// TwinCAT 3 PLC project Projet_Base
// ProgramVersion: 3.1.4026.12
// CompilerDefines: VISU_USEPROPERTYINFO
// libraries:
//   CmpBitmapPool, * (System)
//   Tc2_ControllerToolbox, * (Beckhoff Automation GmbH)
//   Tc2_ModbusRTU, * (Beckhoff Automation GmbH)
//   Tc2_ModbusSrv, * (Beckhoff Automation GmbH)
//   Tc2_SerialCom, * (Beckhoff Automation GmbH)
//   Tc2_Standard, * (Beckhoff Automation GmbH)
//   Tc2_System, * (Beckhoff Automation GmbH)
//   Tc2_TcpIp, * (Beckhoff Automation GmbH)
//   Tc2_Utilities, * (Beckhoff Automation GmbH)
//   Tc3_Database, * (Beckhoff Automation GmbH)
//   Tc3_Module, * (Beckhoff Automation GmbH)
//   BASIC,3.31,OSCAT
// project tree:
//   00_FunctionsBlocks/Beckhoff/AlarmManagement/ FB_HeartBeatMasterBackup.TcPOU, FUN_Alarms_CSV.TcPOU, FUN_ReadAlarm_CSV.TcPOU, ServerCSV.TcDUT, ServerSms.TcDUT, SMS_Server.TcPOU
//   00_FunctionsBlocks/Beckhoff/Annexesfunction/ FB_RestartService.TcPOU, FUN_ConnectVPN.TcPOU, FUN_DisconnectVPN.TcPOU, FUN_GetPublicIp.TcPOU, FUN_PingHost.TcPOU, PRG_RestartPlc.TcPOU
//   00_FunctionsBlocks/Beckhoff/Communication/IEC104/ E_ComState.TcDUT, FB_IEC104ServerAkuo.TcPOU, GVL_Cst.TcGVL, ST_IEC104AkuoParam.TcDUT
//   00_FunctionsBlocks/Beckhoff/Communication/Mail/ FUN_SendMail.TcPOU, ServerMail.TcDUT
//   00_FunctionsBlocks/Beckhoff/Communication/ModbusRTU/ CheckStruct.TcPOU, FB_ModbusRTU.TcPOU, FB_ReadModbusRTU_V2.TcPOU, Sample_ModbusRTU.TcPOU, Struct_InputRTU.TcDUT
//   00_FunctionsBlocks/Beckhoff/Communication/ModbusTCP/ FB_ModbusRead.TcPOU, FB_ModbusReadCoils.TcPOU, FB_ModbusReadInput.TcPOU, FB_ModbusReadInputRegs.TcPOU, FB_ModbusWrite.TcPOU, FB_ModbusWriteMultipleCoils.TcPOU, FB_ModbusWriteSingleCoil.TcPOU, FB_ModbusWriteSingleRegister.TcPOU
//   00_FunctionsBlocks/Beckhoff/Communication/SMS/ FB_DeleteAllSMS.TcPOU, FB_DeleteSMS.TcPOU, FB_Extract_Num_Mes.TcPOU, FB_Login.TcPOU, FB_ReadSMS.TcPOU, FB_SendSMS.TcPOU, ST_SMSDataSetEntry_Read.TcDUT, ST_SMSDataSetEntry_Send.TcDUT
//   00_FunctionsBlocks/Beckhoff/Database/ CheckConfig.TcPOU, PRG_EpochConverter.TcPOU, PRG_TimestructConverter.TcPOU, St_DataHisto.TcDUT, St_DataHisto_Epoch.TcDUT, UnixTimestamp.TcPOU
//   00_FunctionsBlocks/Beckhoff/Database/Firebird/ Firebird_CreateTables.TcPOU, Firebird_InsertBuffer.TcPOU, Firebird_InsertBuffer_vEpoch.TcPOU, Firebird_ReadAlarms.TcPOU, Firebird_RetrieveHDBID.TcPOU, Firebird_SelectBuffer.TcPOU, Firebird_WriteAlarms.TcPOU, LoggerFirebird.TcDUT, St_AlarmsV2.TcDUT
//   00_FunctionsBlocks/Beckhoff/Database/InfluxDb/ InfluxDb_AlarmsManagement.TcPOU, InfluxDb_ReadValues.TcPOU, InfluxDb_WriteAlarms.TcPOU, InfluxDb_WriteStruct.TcPOU, LoggerInfluxDb.TcDUT, ST_InfluxAlarmsInsert.TcDUT, ST_InfluxAlarmsRetrieve.TcDUT
//   00_FunctionsBlocks/Beckhoff/Database/SQLCe/ FB_SQLExpert_InsertBuffer_1.TcPOU
//   00_FunctionsBlocks/Beckhoff/Database/SQLite/ SQLite_CreateDb_V2_1.TcPOU, SQLite_DeleteConfDb_1.TcPOU
//   00_FunctionsBlocks/Beckhoff/DataProcessing/Compress/ FB_CompressFile.TcPOU, FUN_CompressCSV.TcPOU
//   00_FunctionsBlocks/Beckhoff/DataProcessing/Database/ DataBase_V2.TcPOU, FB_DeleteFile.TcPOU, FB_SQLExpert_InsertBuffer.TcPOU, SQLite_CreateDb_V2.TcPOU, SQLite_DeleteConfDb.TcPOU
//   00_FunctionsBlocks/Beckhoff/DataProcessing/ FB_MergeWordsToFloat.TcPOU, FB_MessageDynamique.TcPOU, FB_SplitFloatToWords.TcPOU, FB_WordsToFloat32MLE.TcPOU, FUN_Transpose.TcPOU, MOYENNE.TcPOU, ReplaceAll.TcPOU, SavePersistent.TcPOU
//   00_FunctionsBlocks/Beckhoff/DataProcessing/ReadFile/ FB_Read.TcPOU, FB_ReadCSV.TcPOU
//   00_FunctionsBlocks/Beckhoff/DataProcessing/WriteFile/ CheckStruct_Alarms.TcPOU, FB_CreateDir_V2.TcPOU, FB_WriteFile.TcPOU, FB_Write_CSV.TcPOU, FUN_CreateDir_CSV.TcPOU, LoggerCSV.TcDUT, ST_Journal.TcDUT, ST_ValuesAlarms.TcDUT, ST_ValuesWrite.TcDUT
//   00_FunctionsBlocks/Beckhoff/Fifo/ FB_CommandAlternate.TcPOU, FB_DBDatasetFifo.TcPOU, FB_DBDatasetFifo_1min.TcPOU, FB_SMSDatasetFifo_Read.TcPOU, FB_SMSDatasetFifo_Send.TcPOU, GVL_Fifo.TcGVL
//   00_FunctionsBlocks/Common/AlarmManagement/ FB_AlarmCodeManager.TcPOU, FB_CheckCommand.TcPOU, FB_CheckSetpt.TcPOU, FB_DetectFixedValue.TcPOU, FB_DetectFlicker.TcPOU, FB_UnknownEvent.TcPOU
//   00_FunctionsBlocks/Common/BoolManagement/ FB_CountNinTimeWindow.TcPOU, FB_TapVariable.TcPOU, FB_Toggle2Tap.TcPOU, FB_WordToArrayOfBool.TcPOU, FB_WriteOnChange.TcPOU, RS_NoReset.TcPOU
//   00_FunctionsBlocks/Common/Ctrl/ FB_PIDRegulation.TcPOU
//   00_FunctionsBlocks/Common/DataProcessing/ FB_Average.TcPOU, FB_CountBitOfWordAtTrue.TcPOU, FB_Integrate.TcPOU, FB_MovingAverage.TcPOU, FB_Ramp.TcPOU, FB_Ramp_Time.TcPOU, FB_Smooth.TcPOU, FB_XorWord.TcPOU, Split.TcPOU, Substring.TcPOU
//   00_FunctionsBlocks/Common/DataProcessing/MergeWord/ FB_ISKRA_T5.TcPOU, FB_ISKRA_T6.TcPOU, FB_MergeWordsToDint.TcPOU, FB_MergeWordsToUint.TcPOU, FB_MergeWordsToUlint.TcPOU, FB_WordsToDint64BE.TcPOU
//   00_FunctionsBlocks/Common/DataProcessing/SplitWord/ FB_SplitDintToWords.TcPOU, FB_SplitRealToWords.TcPOU, FB_SplitRealToWords_IEEE754.TcPOU, FB_SplitUlintToWords.TcPOU, FB_SplitWordToByte.TcPOU
//   00_FunctionsBlocks/Common/HistorizationVisu/ FB_OperationIndex.TcPOU, GetTime.TcPOU
//   00_FunctionsBlocks/Templates/ FB_EX_Example.TcPOU
//   01_Equipement_Library/Actuators/ CB_AuxMVCB_Sch.TcDUT, CB_MainMVCB_Sch.TcDUT, CB_Standard.TcDUT, CB_FeederMVCB_Sch.TcDUT, CB_MeasureMVCB_Sch.TcDUT, CB_Switch.TcDUT, FB_CB_AuxMVCB.TcPOU, FB_CB_GridMVCB.TcPOU, FB_CB_MainHVCB.TcPOU, FB_CB_MainMVCB.TcPOU, FB_CB_MeasureMVCB.TcPOU, CB_MainHVCB_Sch.TcDUT, CB.TcDUT, FB_CB_Base.TcPOU, FB_CB_FeederMVCB.TcPOU, FB_CB_MVSwitch.TcPOU, FB_CB_Switch.TcPOU
//   01_Equipement_Library/Batteries/ BAT.TcDUT, BAT_KP.TcDUT, BAT_NARADA.TcDUT, BAT_SAMS.TcDUT, BAT_SAFT.TcDUT, BAT_Standard.TcDUT, FB_BAT_NARADA.TcPOU, FB_BAT_Sams.TcPOU, FB_BAT_Base.TcPOU, FB_BAT_KP_MK1.TcPOU, FB_BAT_Saft.TcPOU, FUN_AlarmManagement_STR.TcPOU, Module.TcDUT, CELL.TcDUT, BMS_SAFT.TcDUT, Rack.TcDUT, RackString_NARADA.TcDUT, RackString_SAFT.TcDUT, RackString.TcDUT, RackString_KP.TcDUT, Rack_SAMS.TcDUT, RackString_SAMS.TcDUT, St_AlarmCodeSamsung.TcDUT
//   01_Equipement_Library/Datalogger/ Datalogger.TcDUT, Datalogger_IOWIT.TcDUT, Datalogger_SchSkid.TcDUT, Datalogger_Secu.TcDUT, Datalogger_SENECA.TcDUT, FB_Datalogger_Base.TcPOU, FB_Datalogger_IOWIT.TcPOU (excluded from build), FB_Datalogger_SchSkid.TcPOU, FB_Datalogger_SENECA.TcPOU (excluded from build), FB_Datalogger_PPCVerrerie.TcPOU (excluded from build), Datalogger_PPCVerrerie.TcDUT (excluded from build)
//   01_Equipement_Library/Fan/ Fan_Standard.TcDUT, Fan.TcDUT, FB_Fan_Basic.TcPOU
//   01_Equipement_Library/FireSystem %28FSS%29/ FSS_Standard.TcDUT (not stored), FB_FSS.TcPOU (not stored), FSS.TcDUT (not stored)
//   01_Equipement_Library/GRID/ FB_GRID_Base.TcPOU, FB_GRID_Enedis.TcPOU, FB_GRID_PLAN.TcPOU, GRID.TcDUT, GRID_MADI.TcDUT, GRID_Enedis.TcDUT, FB_GRID_MADI.TcPOU, GRID_PLAN.TcDUT, IEC104_PLAN.TcDUT, IEC104_MADI.TcDUT
//   01_Equipement_Library/HVAC/ FB_HVAC_MeAcMbs1.TcPOU, FB_HVAC_Standard.TcPOU, FB_HVAC_Base.TcPOU, FB_HVAC_MADI.TcPOU, HVAC.TcDUT, HVAC_MADI.TcDUT, HVAC_MeAcMbs1.TcDUT, HVAC_NARADA.TcDUT, HVAC_Standard.TcDUT, HVAC_SAFT.TcDUT
//   01_Equipement_Library/Inverter/ FB_INV_PE_HEMK.TcPOU, FB_INV_PE_HEMG3.TcPOU, FB_INV_ABB_PVS175TL.TcPOU, FB_SKID_PE_HEMG3.TcPOU, FB_INV_SmaSCXXXXCP_HE.TcPOU, FB_INV_Base.TcPOU, FB_INV_JemaIFX6.TcPOU, FB_INV_Power_One.TcPOU, FB_INV_Sch4400.TcPOU, FB_INV_Huawei_SL.TcPOU, FB_INV_SmaSCXXXXUP_US.TcPOU, FB_INV_Huawei_Sun2000KtlMo.TcPOU, INV.TcDUT, INV_DcModule.TcDUT, INV_DU.TcDUT, INV_ABB_PVS.TcDUT, INV_Huawei.TcDUT, INV_PE_HEMK.TcDUT, INV_PE_HEMG3.TcDUT, SKID_PE_HEMG3.TcDUT, PowerCol_INV_PE_HEMK.TcDUT, PowerCol_INV_PE_HEMG3.TcDUT, INV_SmaSCXXXCP_HE.TcDUT, INV_ClusterPowerOne.TcDUT, INV_Jema_IFX6.TcDUT, INV_PowerOne.TcDUT, INV_Sch4400.TcDUT, INV_SmaSCXXXXUP_US.TcDUT, JuncBox.TcDUT, PowerCol_INV_Jema.TcDUT, PowerCol_INV_JemaAlarms.TcDUT, PowerCol_INV.TcDUT, PowerCol_INV_Power_One.TcDUT, INV_Huawei_SL.TcDUT, STR.TcDUT, STR_SSM.TcDUT
//   01_Equipement_Library/IPC/ FB_IPC.TcPOU, IPC.TcDUT, IPC_Standard.TcDUT
//   01_Equipement_Library/Operation Meter/ FB_PM_ION9200.TcPOU, FB_PM_PM5XXX.TcPOU, FB_PM_Prometer.TcPOU, FB_PM_520x230.TcPOU, FB_PM_A40.TcPOU, FB_PM_Digiware.TcPOU, FB_PM_ION7650.TcPOU, FB_PM_Janitza.TcPOU, FB_PM_PM800.TcPOU, FB_PM_Q100.TcPOU, FB_PM_SM103E.TcPOU, PM.TcDUT, FB_PM_PM3250.TcPOU, PM_DirisA40.TcDUT, PM_ION9200.TcDUT, PM_PM5XXX.TcDUT, PM_Prometer.TcDUT, PM_Standard.TcDUT, PM_PM800.TcDUT, PM_Q100.TcDUT, FB_PM_Base.TcPOU
//   01_Equipement_Library/PCS/ DCInputs_PE.TcDUT, FB_PCS_Base.TcPOU, FB_PCS_Jema_IBX3.TcPOU, FB_PCS_PE.TcPOU, FB_PCS_Sma_SCS3450UP.TcPOU, PCS.TcDUT, PCS_Sma.TcDUT, PCS_Jema_IBX3.TcDUT, PCS_PE.TcDUT, PowerCol_JemaAlarms.TcDUT, PowerCol_Jema.TcDUT, PowerCol.TcDUT, PowerCol_PE.TcDUT
//   01_Equipement_Library/PPC/ FB_PPC_Base.TcPOU, FB_PPC_PE.TcPOU, FB_PPC_SmaKita.TcPOU, PPC.TcDUT, PPC_Sma.TcDUT, PPC_PE.TcDUT
//   01_Equipement_Library/ProtectRelay/ FB_ProtectRelay_DM2.TcPOU, FB_ProtectRelay_Flair23DM.TcPOU, FB_ProtectRelay_MaxI.TcPOU, FB_ProtectRelay_Micom.TcPOU, FB_ProtectRelay_NSXCB.TcPOU, FB_ProtectRelay_PACE100ST.TcPOU, FB_ProtectRelay_REF615.TcPOU, FB_ProtectRelay_SchP3U30.TcPOU, FB_ProtectRelay_SepamT20.TcPOU, FB_ProtectRelay_Siprotec.TcPOU, FB_ProtectRelay_SMNS7SL86.TcPOU, FB_ProtectRelay_VIP410.TcPOU, FB_ProtectRelay_WIP1.TcPOU, FB_ProtectRelay_SEPAM10a.TcPOU, FB_ProtectRelay_Base.TcPOU, FB_ProtectRelay_SepamS48.TcPOU, ProtectRelay_Micom.TcDUT, ProtectRelay_SchP30U30.TcDUT, ProtectRelay_Siprotec.TcDUT, ProtectRelay_SMNS7L86.TcDUT, ProtectRelay_Standard.TcDUT, ProtectRelay_Flair23DM.TcDUT, ProtectRelay_NSXCB.TcDUT, ProtectRelay_PACE100ST.TcDUT, ProtectRelay_REFIO.TcDUT, ProtectRelay.TcDUT, ProtectRelay_S42.TcDUT, ProtectRelay_S48.TcDUT, ProtectRelay_T20.TcDUT, ProtectRelay_T87.TcDUT, ProtectRelay_VIP410.TcDUT, ProtectRelay_WIP1.TcDUT
//   01_Equipement_Library/Router/ FB_Router.TcPOU, Router.TcDUT, Router_Standard.TcDUT
//   01_Equipement_Library/Sensors/ANA/ ANA.TcDUT, ANA_DevStd_Prom.TcDUT, ANA_DustIQ.TcDUT, ANA_Standard.TcDUT, FB_ANA_Base.TcPOU, FB_ANA_IO.TcPOU, FB_ANA_Irra_Fx.TcPOU
//   01_Equipement_Library/Sensors/COM/ AllInOne.TcDUT, AllInOne_Standard.TcDUT, DustIQ.TcDUT, DustIQ_Standard.TcDUT, FB_ANA_AllInOne.TcPOU, FB_ANA_DustIQ.TcPOU, FB_ANA_SMP1X.TcPOU, PV_temp_sensor.TcDUT, SMP1X.TcDUT
//   01_Equipement_Library/Sensors/TOR/ FB_TOR_CB.TcPOU, FB_TOR_Digicode.TcPOU, FB_TOR_Standard.TcPOU, FB_TOR_ES.TcPOU, FB_TOR_Fuse.TcPOU, FB_TOR_MS.TcPOU, FB_TOR_Spd.TcPOU, FB_TOR_VP.TcPOU, TOR.TcDUT, FB_TOR_Base.TcPOU, FB_TOR_DS.TcPOU, FB_TOR_Rain.TcPOU, FB_TOR_SD.TcPOU, FB_TOR_ToS.TcPOU, TOR_CB.TcDUT, TOR_Standard.TcDUT, TOR_Rain.TcDUT
//   01_Equipement_Library/TAC/ FB_TAC.TcPOU, TAC.TcDUT, TAC_Standard.TcDUT
//   01_Equipement_Library/Tariff Meter/ EM_ION8650.TcDUT, EM_Standard.TcDUT, FB_EM_Base.TcPOU, FB_EM_ION8650.TcPOU, FB_EM_Pulse.TcPOU, EM.TcDUT
//   01_Equipement_Library/Tracker/ FB_NCU_Base.TcPOU, FB_NCU_Axial.TcPOU, NCU.TcDUT, NCU_Axial.TcDUT, TRK.TcDUT, TRK_Axial.TcDUT
//   01_Equipement_Library/Transfo/ FB_Transfo_Base.TcPOU, FB_Transfo_HVCom.TcPOU, FB_Transfo_MV.TcPOU, FB_Transfo_MVCom.TcPOU, TapChanger.TcDUT, Transfo.TcDUT, Transfo_HV.TcDUT, Transfo_MV.TcDUT
//   01_Equipement_Library/UPS/ FB_UPS_MCSU4.TcPOU, FB_UPS_PS10048.TcPOU, UPS_CXC.TcDUT, FB_UPS_CXC.TcPOU, FB_UPS_Base.TcPOU, FB_UPS_Eneris.TcPOU, UPS.TcDUT, UPS_Eneris.TcDUT, UPS_MCSU4.TcDUT, UPS_PS10048.TcDUT
//   02_Product_Library/EnergyStorageSystem%28ESS%29/ ESS_BARD.TcDUT (not stored), ESS_Exd.TcDUT (not stored), ESS_MADI.TcDUT (not stored), ESS_NARADA.TcDUT (not stored), FB_ESS_MADI.TcPOU (not stored), FB_ESS_BARD.TcPOU (not stored), FB_ESS_Base.TcPOU (not stored), FB_ESS_NARADA.TcPOU (not stored), FB_ESS.TcPOU (not stored), ESS.TcDUT (not stored)
//   02_Product_Library/PowerTRansformerStation%28PTR%29/ FB_PTR.TcPOU (not stored), FB_PTR_Base.TcPOU (not stored), PTR_Exd.TcDUT (not stored), PTR.TcDUT (not stored)
//   02_Product_Library/Substation%28SUB_MV%29/ FB_SUBMV.TcPOU (not stored), FB_SUBMV_Base.TcPOU (not stored), SUBMV.TcDUT (not stored), SUBMV_Exd.TcDUT (not stored)
//   02_Product_Library/Substation%28SUB_HV%29/ FB_SUBHV.TcPOU (not stored), FB_SUBHV_Base.TcPOU (not stored), SUBHV.TcDUT (not stored), SUBHV_Exd.TcDUT (not stored)
//   02_Product_Library/Trackers%28TRK%29/ FB_TRKCtl.TcPOU (not stored), TRKCtl.TcDUT (not stored)
//   02_Product_Library/WeatherStation %28WS%29/ FB_WS.TcPOU (not stored), FB_WS_Base.TcPOU (not stored), WS.TcDUT (not stored), WS_RAV2.TcDUT (not stored)
//   03_Power_Plant %28PP%29/ FB_PP.TcPOU (not stored), PP.TcDUT (not stored)
//   04_Application/ALARM/ FUN_Alarms.TcPOU, Redundancy.TcPOU
//   04_Application/Annexes_Functions/ PRG_AnnexesFunctions.TcPOU
//   04_Application/BDD/ FUN_Write_CSV.TcPOU
//   04_Application/Checks/ CheckBounds.TcPOU, CheckDivDInt.TcPOU, CheckDivLInt.TcPOU, CheckDivLReal.TcPOU, CheckDivReal.TcPOU, CheckLRangeSigned.TcPOU, CheckLRangeUnsigned.TcPOU, CheckPointer.TcPOU, CheckRangeSigned.TcPOU, CheckRangeUnsigned.TcPOU
//   04_Application/COM/ COM_Status.TcDUT, ModbusTcp.TcPOU
//   04_Application/CONFIG/ GVL_BASE.TcGVL, GVL_Beckhoff.TcGVL, GVL_CFG.TcGVL, GVL_Check.TcGVL, GVL_DataBaseStructures.TcGVL
//   04_Application/EMS/ EMS.TcDUT, IN_EMS.TcDUT, OUT_EMS.TcDUT, PRG_EMS.TcPOU
//   04_Application/HMI/BESS/ BESS_HMI.TcPOU
//   04_Application/HMI/ HMI.TcPOU
//   04_Application/HMI/HPP/ HPP_HMI.TcPOU
//   04_Application/HMI/Infos/ InfosIO.TcPOU
//   04_Application/HMI/Parameters/ ParamBESS_HMI.TcPOU, ParamEMS.TcPOU
//   04_Application/HMI/SPP/ SPP_HMI.TcPOU
//   04_Application/IO/ IO.TcDUT, PRG_IO.TcPOU, ST_AI.TcDUT, ST_AO.TcDUT, ST_DI.TcDUT, ST_DO.TcDUT
//   04_Application/MAIN/ MAIN.TcPOU, POU.TcPOU, TEST.TcPOU
//   04_Application/OPC/ AllAlarms.TcDUT, AllDataR.TcDUT, OPCAlarms.TcDUT, AllDataWPulse.TcDUT, AllDataWToggle.TcDUT, AllValueW.TcDUT, OpcUa.TcPOU
//   / AnnexFunction.TcTTO, PlcTask.TcTTO
// real-time tasks:
//   TASK PlcTask: cycle T#10ms, priority 8, ADS port 350
//   TASK Emul_Task: cycle T#25000us, priority 16, ADS port 351
//   TASK Database_Task: cycle T#100000us, priority 14, ADS port 352
//   TASK IOTask: cycle T#10ms, priority 6, ADS port 301
//   TASK AnnexFunction: cycle T#100000us, priority 10, ADS port 353
// I/O:
//   DEVICE Périphérique 1 (EtherCAT) (disabled), AmsNetId 192.168.13.104.2.1
//     Terme 1 (EK1200) [EK1200-5000 EtherCAT Power supply (2A E-Bus)]
//       Terme 2 (EL4024) [EL4024 4Ch. Ana. Output 4-20mA, 12bit]
//       Terme 3 (EL3024) [EL3024 4Ch. Ana. Input 4-20mA DIFF]
//       Terme 4 (EL9011) [EL9011 End Terminal]

CONFIGURATION Projet_Base
    RESOURCE PLC ON TwinCAT3
        TASK AnnexFunction(INTERVAL := T#100000us, PRIORITY := 10);
        TASK PlcTask(INTERVAL := T#10ms, PRIORITY := 8);
        PROGRAM PRG_AnnexesFunctions WITH AnnexFunction : PRG_AnnexesFunctions;
        PROGRAM MAIN WITH PlcTask : MAIN;
    END_RESOURCE
END_CONFIGURATION

// ---- 00_FunctionsBlocks/Beckhoff/AlarmManagement/ServerCSV.TcDUT

TYPE ServerCSV :
STRUCT
	FileSize			: ULINT;			(*(o) Size of the file being used for logging alarms *)
	TimeCreation		: TIMESTRUCT;		(* TimeCreation of file*)
	TimeModif			: TIMESTRUCT;		(* Time Modif of file*)
	MesAlarmCode		: WORD;				(* Alarm Code related to this functionnality*)

END_STRUCT
END_TYPE

// ---- 00_FunctionsBlocks/Beckhoff/AlarmManagement/ServerSms.TcDUT

TYPE ServerSms :
STRUCT
	NbrUtiliActive			: INT;									(* Number of users*)
	MesAlarmCode			: WORD;									(* Alarm Code*)
	AX_Numtel				: ARRAY[1..CstNbUser] OF STRING(26);	(*Tel Number list*)
	AX_Subscribed			: ARRAY[1..CstNbUser] OF BOOL;			(*Subscription list*)
	AX_NomUtili				: ARRAY[1..CstNbUser] OF STRING(50); 	(* User name list	*)
	AX_UserLVL				: ARRAY[1..CstNbUser] OF WORD; 		(*User Level*)

END_STRUCT
END_TYPE

// ---- 00_FunctionsBlocks/Beckhoff/Communication/IEC104/E_ComState.TcDUT
TYPE E_ComState :
(
	INIT := 0,
	IDLE,
	CONNECT,
	DATATRANSFER,
	DISCONNECT
);
END_TYPE

// ---- 00_FunctionsBlocks/Beckhoff/Communication/IEC104/ST_IEC104AkuoParam.TcDUT
TYPE ST_IEC104AkuoParam :
STRUCT
	bEnableFlicker 	: BOOL :=  TRUE ;
	tFlickerWindow	: TIME := T#10S ; 
	uFlickerNumber	: UINT := 7  ; 

	iLocalPort 		: UDINT := 2404;						// locl port
	sLocalHost		: STRING := '127.0.0.1'; 			// server IP address. 
	iAOnb			: INT ;								// Number of AO being treated ( <GVL_Cst.CstNbAOEntries)
 
END_STRUCT
END_TYPE

// ---- 00_FunctionsBlocks/Beckhoff/Communication/Mail/ServerMail.TcDUT

TYPE ServerMail :
STRUCT

	MesAlarmCode			: WORD;			(*alarm code *)
	
	AX_MailAddr				: ARRAY[1..CstNbUser] OF STRING(255);		(* Mail Address List*)
	AX_Subscribed			: ARRAY[1..CstNbUser] OF BOOL;				(* Mail subscription list*)
	AX_NomUtili				: ARRAY[1..CstNbUser] OF STRING(50); 		(* User Name List*)
	AX_UserLVL				: ARRAY[1..CstNbUser] OF WORD; 		(* User Level*)
	
	OUT_NbMailSent			: ULINT;									(* Number of mail being sent *)
	
END_STRUCT
END_TYPE

// ---- 00_FunctionsBlocks/Beckhoff/Communication/ModbusRTU/Struct_InputRTU.TcDUT
TYPE Struct_InputRTU :
STRUCT
	InStartAddr			: WORD;
	InQuantity			: WORD;
	InUnitID			: BYTE;
	InBuffer			: POINTER TO BYTE;
	InFunction			: UINT;
	OutBusy				: POINTER TO BOOL;
	OutError			: POINTER TO BOOL;
	OutCompleted 		: POINTER TO BOOL;
	OutErrorId			: POINTER TO INT ; 
END_STRUCT
END_TYPE

// ---- 00_FunctionsBlocks/Beckhoff/Communication/SMS/ST_SMSDataSetEntry_Read.TcDUT
TYPE ST_SMSDataSetEntry_Read :
STRUCT
	Message : STRING(160);  // Commande envoyé par message
	Num		: STRING(20);  //  Numéro de l'utilisateur
END_STRUCT
END_TYPE

// ---- 00_FunctionsBlocks/Beckhoff/Communication/SMS/ST_SMSDataSetEntry_Send.TcDUT
TYPE ST_SMSDataSetEntry_Send :
STRUCT
	ID				: UINT;			// Unic ID to identify the alarm
	IndexWord		: UINT; 		//Index du word correspondant aux alarmes
	IndexBit		: UINT; 		//Index du bit correspondant a l'alarme
	Active			: BOOL; 		//Ne pas remplir - Utilisé par le code
	Num_tel			: STRING(20);//Ne pas remplir - Utilisé par le code
	TimeStamp_Act	: STRING;	// TimeStamp of the last activation or desactivation
	Alarms_LVL		: WORD;
END_STRUCT
END_TYPE

// ---- 00_FunctionsBlocks/Beckhoff/Database/Firebird/LoggerFirebird.TcDUT

TYPE LoggerFirebird :
STRUCT
	MesAlarmCode		: WORD;				// Alarm Code

END_STRUCT
END_TYPE

// ---- 00_FunctionsBlocks/Beckhoff/Database/Firebird/St_AlarmsV2.TcDUT
TYPE St_AlarmsV2 :
STRUCT
	TIMESTAMP_START : DT;
	TIMESTAMP_STOP	: DT;
	ALARMSID 		: DINT;
	ACT				: INT;
	ACK				: INT;
	

END_STRUCT
END_TYPE

// ---- 00_FunctionsBlocks/Beckhoff/Database/InfluxDb/LoggerInfluxDb.TcDUT
TYPE LoggerInfluxDb :
STRUCT
	MesAlarmCode		: WORD;				// Alarm Code
END_STRUCT
END_TYPE

// ---- 00_FunctionsBlocks/Beckhoff/Database/InfluxDb/ST_InfluxAlarmsInsert.TcDUT
TYPE ST_InfluxAlarmsInsert :
STRUCT
    {attribute 'TagName' := 'Message'}
	Message		 	: T_MaxString;	// Alarm Message 
    {attribute 'FieldName' := 'ID'}	
	ID			: 	ULINT;
    {attribute 'FieldName' := 'Value'}	
	Value 		: BOOL;
    {attribute 'FieldName' := 'Ack'}	
	Ack			: BOOL;	
END_STRUCT
END_TYPE

// ---- 00_FunctionsBlocks/Beckhoff/Database/InfluxDb/ST_InfluxAlarmsRetrieve.TcDUT
TYPE ST_InfluxAlarmsRetrieve :
STRUCT
    {attribute 'TagName' := 'time'}
	MesTime			: LINT;
    {attribute 'TagName' := 'Message'}
	Message		 	: T_MaxString;	// Alarm Message 
    {attribute 'FieldName' := 'ID'}	
	ID				: ULINT;
    {attribute 'FieldName' := 'Value'}	
	Value 			: BOOL;
    {attribute 'FieldName' := 'Ack'}	
	Ack				: BOOL;	
END_STRUCT
END_TYPE

// ---- 00_FunctionsBlocks/Beckhoff/Database/St_DataHisto.TcDUT
TYPE St_DataHisto :
STRUCT
	Timestamp		: TIMESTRUCT;
	ParentId		: DINT;
	Value			: LREAL;
END_STRUCT
END_TYPE

// ---- 00_FunctionsBlocks/Beckhoff/Database/St_DataHisto_Epoch.TcDUT
TYPE St_DataHisto_Epoch :
STRUCT
	Timestamp		: ULINT;
	ParentId		: DINT;
	Value			: LREAL;
END_STRUCT
END_TYPE

// ---- 00_FunctionsBlocks/Beckhoff/DataProcessing/WriteFile/LoggerCSV.TcDUT

TYPE LoggerCSV :
STRUCT
	FileSize			: ULINT;			(* (o) File size *)
	TimeCreation		: TIMESTRUCT;		(* TimeCreation of file*)
	TimeModif			: TIMESTRUCT;		(* Time Modif of file*)
	MesAlarmCode		: WORD;				(* Alarm Code*)

END_STRUCT
END_TYPE

// ---- 00_FunctionsBlocks/Beckhoff/DataProcessing/WriteFile/ST_Journal.TcDUT
TYPE ST_Journal :
STRUCT
	Message			: STRING(150); //Message texte à envoyer aux utilisateurs
	Groupe			: (Sans_Operation,Avec_Operation_Act,Avec_Operation_Act_Des):=1; // 0:sans action,1:Envois sms sur acttivation,2:Envois sms sur activation et desactivation
	Ax_ParamB		: ARRAY [1..4] OF POINTER TO BOOL; //Tableau boolean permettant d'envoyer un message dynamique.
	Ax_ParamI		: ARRAY [1..4] OF POINTER TO SINT; //Tableau Sint permettant d'envoyer un message dynamique.
END_STRUCT
END_TYPE

// ---- 00_FunctionsBlocks/Beckhoff/DataProcessing/WriteFile/ST_ValuesAlarms.TcDUT
TYPE ST_ValuesAlarms :
STRUCT
	ID				: UINT;		// Unic ID to identify the alarm 
	Message		 	: STRING(160);	// Alarm Message 
	Value 			: BOOL;		// Value of the alarm
	Ack 			: BOOL;		// Ack of the alarm	
	TimeStamp_Act	: STRING;	// TimeStamp of the last activation or desactivation
	
	Groupe			: UINT:=0; // 0:sans action,1:Envois sms sur acttivation,2:Envois sms sur activation et desactivation
	Alarms_LVL		: WORD:=1; // Si Num utilisateur > Alarms_LVL alors il ne recoit pas les sms 1 := Standart , 2 := Syntehses , 3:= Securité
END_STRUCT
END_TYPE

// ---- 00_FunctionsBlocks/Beckhoff/DataProcessing/WriteFile/ST_ValuesWrite.TcDUT
TYPE ST_ValuesWrite :
STRUCT
	Description : STRING;
	Address 	: POINTER TO REAL;
	AddressLR	: POINTER TO LREAL;
	AddressUL	: POINTER TO ULINT;
	AddressUI	: POINTER TO UINT;
	Size		: UINT;
	Sampling	: DINT := 1000;		// Period of sampling
	
END_STRUCT
END_TYPE

// ---- 01_Equipement_Library/Actuators/CB_AuxMVCB_Sch.TcDUT
///////////
// Structure For Bousquet. Main Operating Data to be saved (ex: OPC).  
//////////

TYPE CB_AuxMVCB_Sch :
STRUCT
	//DI
	MesData					: CB ;      (* Object*)
	MesFuseBurned		    : BOOL ; 	(* The Fuse is burned*)
	MesEarth				: BOOL ; 	(* The Cell is grounded*)
	MesLvSwitch				: BOOL ; 	(* LV switch gear PT1 delivery station is closed closed*)
	MesUpstream_Switch		: BOOL ; 	(* Upstream swit is closedch gear closed *)
	MesAlim_48v				: BOOL ; 	(*  is closed48V switch gear closed*)


END_STRUCT
END_TYPE

// ---- 01_Equipement_Library/Actuators/CB_MainMVCB_Sch.TcDUT
///////////
// Structure for MainMVCB Schneider. Main Operating Data to be saved (ex: OPC).  
//////////

TYPE CB_MainMVCB_Sch :
STRUCT
	//DI
	MesData					: CB   ;    (* Object*)
	MesComutLocal		    : BOOL ; 	(* The cell selector is in local position*)
	MesAlarmPwr		        : BOOL ; 	(* The cell motorization has a power supply fault*)
	MesEarth				: BOOL ; 	(* The cell is grounded (earthing)*)
	MesTripped	    	    : BOOL ; 	(* The cell is tripped (opened and locked due to alarm)*)
	OUT_CmdOpen				: BOOL ; 	(* The SCADA sends an Open command to the cell*)
	OUT_CmdClose			: BOOL ; 	(* The SCADA sends a Close command to the cell*)
	MesOpened_Sect			: BOOL ; 	(* The associated switchgear is opened*)
	

	MesSwitchG				: BOOL ;    (* Plant switch gear     *)
	MesTest_Serv 			: BOOL ;	(* test/service          *)
	MesDefaulr_48VCC		: BOOL ;    (* 48Vcc default         *)
	
	
	
END_STRUCT
END_TYPE

// ---- 01_Equipement_Library/Actuators/CB_Standard.TcDUT
TYPE CB_Standard :
///////////
// Structure For Bousquet. Main Operating Data to be saved ( ex: OPC )   
//////////
STRUCT
	//DI
	MesData				: CB ;  (* Object*)

END_STRUCT
END_TYPE

// ---- 01_Equipement_Library/Actuators/CB_FeederMVCB_Sch.TcDUT
///////////
// Structure For Bousquet . Main Operating Data to be saved (ex: OPC).  
//////////

TYPE CB_FeederMVCB_Sch :
STRUCT
	//DI
	MesData					: CB   ;    (* Object*)
	MesComutLocal		    : BOOL ; 	(* The cell selector is in local position*)
	MesAlarmPwr		        : BOOL ; 	(* The cell motorization has a power supply fault*)
	MesEarth				: BOOL ; 	(* The cell is grounded (earthing)*)
	MesTripped	    	    : BOOL ; 	(* The cell is tripped (opened and locked due to alarm)*)
	OUT_CmdOpen				: BOOL ; 	(* The SCADA sends an Open command to the cell*)
	OUT_CmdClose			: BOOL ; 	(* The SCADA sends a Close command to the cell*)
	MesOpened_Sect			: BOOL ;    (* The associated switchgear is opened*)
	
END_STRUCT
END_TYPE

// ---- 01_Equipement_Library/Actuators/CB_MeasureMVCB_Sch.TcDUT
///////////
// Structure For Bousquet. Main Operating Data to be saved (ex: OPC).  
//////////

TYPE CB_MeasureMVCB_Sch :
STRUCT
	//DI
	MesData					: CB ;      (* Object*)
	MesFuseBurned		    : BOOL ; 	(* The Fuse is burned*)
	MesEarth				: BOOL ; 	(* The Cell is grounded*)

END_STRUCT
END_TYPE

// ---- 01_Equipement_Library/Actuators/CB_Switch.TcDUT
///////////
// Structure For Bousquet . Main Operating Data to be saved (ex: OPC).  
//////////

TYPE CB_Switch :
STRUCT
	//DI
	MesData					: CB   ;    (* Object*)
	MesAlarmPwr		        : BOOL ; 	(* The cell motorization has a power supply fault*)

	OUT_CmdOpen				: BOOL ; 	(* The SCADA sends an Open command to the cell*)
	OUT_CmdClose			: BOOL ; 	(* The SCADA sends a Close command to the cell*)
	
END_STRUCT
END_TYPE

// ---- 01_Equipement_Library/Actuators/CB_MainHVCB_Sch.TcDUT
///////////
// Structure For Bousquet . Main Operating Data to be saved (ex: OPC).  
//////////

TYPE CB_MainHVCB_Sch :
STRUCT
	//DI
	MesData					: CB   ;    (* Object*)
	MesComutLocal		    : BOOL ; 	(* The cell selector is in local position*)
	MesAlarmPwr		        : BOOL ; 	(* The cell motorization has a power supply fault*)
	MesEarth				: BOOL ; 	(* The cell is grounded (earthing)*)
	MesTripped	    	    : BOOL ; 	(* The cell is tripped (opened and locked due to alarm)*)

	MesAlarm_SF6      			: BOOL ; (* Not enough SF6 gaz *)
	MesAlarm_Disarmed      		: BOOL ; (* HVCB Command is disarmed*)
	MesAlarm_ArmingMotor   		: BOOL ; (* Arming motorization is on fault*)
	MesAlarm_230V  		 		: BOOL ; (* 230V Aux is on fault*)
	MesOpened_Sect				: BOOL ; (* The associated switchgear is opened*)
	
END_STRUCT
END_TYPE

// ---- 01_Equipement_Library/Actuators/CB.TcDUT
TYPE CB :
///////////
// Structure For Bousquet. Main Operating Data to be saved ( ex: OPC )   
//////////
STRUCT
	//DI
	MesClosed		: BOOL ;	(* Cell is closed*)
	MesOpened		: BOOL ;	(* cell is opened*)
	
	MesAlarmCode	: WORD ;	(* Internal Akuo Alarm Code*)
	MesWarningCode	: WORD ;	(* Internal Akuo Warning Code*)
	MesEventCode	: WORD ;	(* Internal Akuo Warning Code*)
	
	MesCP_Open		: BOOL ;   	(* Cal(NA) Permanent Conditions*)
	MesCP_Close		: BOOL ; 	(* Cal(NA) Permanent Conditions*) 

END_STRUCT
END_TYPE

// ---- 01_Equipement_Library/Batteries/BAT.TcDUT
///////////
// Structure For Battery Controller. Main Operating Data to be saved ( ex: OPC ) .  
//////////

TYPE BAT :
STRUCT

	MesEnomConnected			: REAL ; 		(* (kWh) Nameplate Energy Capacity [WHRtg]          *)      	

	MesIdc						: REAL;			(* (A) Summation of all racks*)
	MesUdc						: REAL;			(* (V) Voltage of the rack, average*)

	MesSoC						: REAL; 		(* (%) SoC Average (not including racks with protection).*)
	MesSoH						: REAL; 		(* (%) SoH Average*)
	MesDoD						: REAL;			(* (%) Depth of Discharge*)

	MesCCL						: REAL;			(* (A) Charge Current Limit*)
	MesDCL						: REAL;			(* (A) Discharge Current Limit*)
	MesCPL						: REAL ; 		(* (kW) Charge Power Limit - To zero if Estop is set . *)
	MesDPL						: REAL ; 		(* (kW) Discharge Power Limit - To zero if Estop is set .*)
	MesECharge					: REAL ; 		(* (kWh) Total Energy charged over time *)
	MesEDischarge				: REAL ; 		(* (kWh) Total Energy Discharge over time *)

	ParamNbRacks				: UINT ; 		(* Number of racks set in BBMS*)
	ParamNbModule				: UINT ; 		(* Number of modules per strings set in BBMS *)
	ParamStringNbMin			: UINT ; 		(* Minimal number of strings Operable in order to works set at BBMS *)
	ParamUdiff					: REAL ;		(* Maximum voltage difference between  string for connexion set in BBMS . *)
	
// Evaluate	
	MesEconnected 				: REAL; 		(* Energy available for charge / discharge in the system BBMS. *)
	MesNbRackNormal				: UINT; 		(* Number of racks without alarms. *)
	MesPdc						: REAL; 		(*(kW) DC Power*)

	MesIDState              	: WORD; 			(* (NA) State of the Battery Bank [State]          *)
	MesEvt1						: DWORD;
    MesEvtVnd1					: DWORD;                	                
	MesAlarmCode				: WORD;			(* (NA) Internal Akuo AlarmCode*)
	
	MesEventCode				: WORD;			(* (NA) Internal Akuo EventCode	*)
	MesAlarmCode_MesEvt1_1		: WORD;
	MesAlarmCode_MesEvt1_2		: WORD;
	
	MesAlarmCode_MesEvtVnd1_1	: WORD;
	MesAlarmCode_MesEvtVnd1_2	: WORD;
	MesWarningCode				: WORD;			(* (NA) Internal Akuo WarningCode*)
	
	MesState					: WORD; 		(* (NA) State of the Bat*)
	MesSoC_Min					: REAL;			(* (%) Minimal SoC of rack*)
	MesSoC_Max					: REAL;			(* (%) Maximal SoC of rack*)
	MesSoC_Max_memory			: REAL ;		(* (%) Maximal SoC reached memory*)
	MesAlarmCom					: BOOL ;		(* Communication alarm*)
	MesWarningCom				: BOOL ;		(* Communication warning*)
	
	
	
	MesCP_Read					: BOOL := TRUE;		(* Read function enable *)
	MesCP_Write					: BOOL ;		(* Write function enable *)
	
	
END_STRUCT
END_TYPE

// ---- 01_Equipement_Library/Batteries/BAT_KP.TcDUT
{attribute 'pack_mode' := '1'}

TYPE BAT_KP :
STRUCT
	MesData						: BAT;			(* Base model*)

	MesSoCConnected				: REAL; 		(* (%) SoC Connected (not including racks with protection).*)

	MesNbCellbalancing				: WORD	; (*(NA) Battery Cell Balancing Count [NCellBal]            *)
	MesNbCycle						: UINT  ; (* (NA) Number of cycles*)
	MesChargeStatus					: UINT  ; (* (NA) Charge status*)
	MesTypeBattery					: WORD  ; (* (NA) Type of battery read on BMS*)
	MesNbRackTot					: WORD	; (*(NA) String Count [NStr]                         		*)
	MesRemoteControl				: BOOL  ; (* (NA) is remote control active on battery system		*)
	MesNbRackConnected              : WORD	; (*(NA) Connected String Count [NStrCon]                   *)

	
	MesIdcMax_Rack                  : REAL  ; (*(A) Max String Current [StrAMax]                        *)
	MesIDRack_Imax_Rack             : WORD	; (*(NA) Max String Current String [StrAMaxStr]             *)
	MesIdcMin_Rack                  : REAL  ; (*(A) Min String Current [StrAMin]                        *)
	MesIDRack_Imin_Rack             : WORD	; (*(NA) Min String Current String [StrAMinStr]             *)

	MesIdc_Rack                     : REAL  ; (*(A) Average String Current [StrAAvg]                    *)


	MesTempMax_Module               : REAL  ; (*(C) Max Module Temperature [ModTmpMax]                  *)
	MesIDRack_TempMax_Module        : WORD	; (*(NA) Max Module Temperature String [ModTmpMaxStr]       *)
	MesIDModule_TempMax_Module      : WORD	; (*(NA) Max Module Temperature Module [ModTmpMaxMod]       *)

	MesTempMin_Module               : REAL  ; (*(C) Min Module Temperature [ModTmpMin]                  *)
	MesIDRack_TempMin_Module        : WORD	; (*(NA) Min Module Temperature String [ModTmpMinStr]       *)
	MesIDModule_TempMin_Module      : WORD	; (*(NA) Min Module Temperature Module [ModTmpMinMod]       *)
	MesTemp_Module                  : REAL  ; (*(C) Average Module Temperature [ModTmpAvg]              *)

	
	MesUdcMax_Cell          		: REAL ; (* (V) Max Cell Voltage [CellVMax]                  *)
	MesIDRack_UdcMax_Cell   		: WORD ; (* (NA) Max Cell Voltage String [CellVMaxStr]       *)
	MesIDModule_UdcMax_Cell 		: WORD ; (* (NA) Max Cell Voltage Module [CellVMaxMod]       *)
	MesUdcMin_Cell          		: REAL ; (* (V) Min Cell Voltage [CellVMin]                  *)
	MesIDRack_UdcMin_Cell   		: WORD ; (* (NA) Min Cell Voltage String [CellVMinStr]       *)
	MesIDModule_UdcMin_Cell 		: WORD ; (* (NA) Min Cell Voltage Module [CellVMinMod]       *)

	
	MesUdcMax_Rack          		: REAL ; (* (V) Max String Voltage [StrVMax]                  *)
	MesIDRack_UdcMax_Rack   		: WORD ; (* (NA) Max Cell Voltage String [StrVMaxStr]       *)
	MesUdcMin_Rack          		: REAL ; (* (V) Min Cell Voltage [StrVMin]                  *)
	MesIDRack_UdcMin_Rack   		: WORD ; (* (NA) Min Cell Voltage String [StrVMinStr]       *)
	MesUdc_Rack						: REAL ;	(* (V) Voltage of the cells, average [StrVAvg]*)


	MesChargeNom					: REAL ; (* (Ah) Nameplate Charge Capacity [AHRtg]          	*)
	     
	MesHeartbeat             		: WORD ; (* (NA) Battery Heartbeat [Hb]                      *)
	MesIDAlarm              		: DWORD ; (* (NA) Battery Event 1 Bitfield [Evt1]             *)                        	

	AX_RACK							: ARRAY[1..CstNbRack_BAT_G] OF RackString_KP;
END_STRUCT
END_TYPE

// ---- 01_Equipement_Library/Batteries/BAT_NARADA.TcDUT
{attribute 'pack_mode' := '1'}

TYPE BAT_NARADA :
STRUCT
	
	MesData							: BAT;	  	(* 	Base model													*)

	MesIDState2             		: REAL  ;   (* ID state pour le alarmManagement des batteries *)
	MesSoCConnected					: REAL  ; 	(* 	(%) SoC Connected (not including racks with protection).	*)
	MesNbRackConnected				: UINT;		(* (NA) Nb of Racks in service ( strings ) 						*)
	MesChargeStatus					: WORD;
	
	// Current                                                                                                       	
	                                                                                                        	
	MesIdcMax_Rack                  : REAL  ; (*	(A) Max String Current [StrAMax]                        	*)
	MesIDRack_Imax_Rack             : WORD	; (*	(NA) Max String Current String [StrAMaxStr]             	*)
	MesIdcMin_Rack                  : REAL  ; (*	(A) Min String Current [StrAMin]                        	*)
	MesIDRack_Imin_Rack             : WORD	; (*	(NA) Min String Current String [StrAMinStr]             	*)
                                                                                                            	
	MesIdc_Rack                     : REAL  ; (*	(A) Average String Current [StrAAvg]                    	*)
	
	MesIdiff						: REAL  ; (* 	(A) 														*)
	
    //Temp      
                                                                                                     	                                                                                            	
	MesTempMax_Cell               	: REAL 	; (*	(℃) Max Cell Temperature [CellTmpMax]             		   	*)
	MesIDRack_TempMax_Cell	        : WORD	; (*	(NA) Max Cell Temperature String [CellTmpMaxStr]       		*)
	MesIDModule_TempMax_Cell	    : WORD	; (*	(NA) Max Cell Temperature Module [CellTmpMaxMod]     	  	*)
    MesIDCell_TempMax			    : WORD	; (*	(NA) Max Cell Temperature [CellTmpMax]	     	  			*)
                                            	                                                        	
	MesTempMin_Cell              	: REAL	; (*	(℃) Min Cell Temperature [CellTmpMin]               	  	*)
	MesIDRack_TempMin_Cell          : WORD	; (*	(NA) Min Cell Temperature String [CellTmpMinStr]       		*)
	MesIDModule_TempMin_Cell        : WORD	; (*	(NA) Min Cell Temperature Module [CellTmpMinMod]       		*)
	MesIDCell_TempMin			    : WORD	; (*	(NA) Max Cell Temperature [CellTmpMin]	     	  			*)
	
	MesTemp_Racks                   : REAL  ; (*	(℃) Average Rals Temperature [RckTmpAvg]             	 	*)
    
	//Voltage         
	
		MesUdiff						: REAL ; (* 	(V) 													*)
	                                                                                                            
		//Cell                                                                                                  
                                                                              	                                
		MesUdcMax_Cell          		: REAL ; (* 	(V) Max Cell Voltage [CellVMax]                 		*)
		MesIDRack_UdcMax_Cell   		: WORD ; (* 	(NA) Max Cell Voltage String [CellVMaxStr]      		*)
		MesIDModule_UdcMax_Cell 		: WORD ; (* 	(NA) Max Cell Voltage Module [CellVMaxMod]      		*)
		MesIDCell_UdcMax		 		: WORD ; (* 	(NA) Max Cell Voltage [CellVMaxMod]      				*)
		                                                                                                        
		                                                                                                        
		MesUdcMin_Cell          		: REAL ; (* 	(V) Min Cell Voltage [CellVMin]                 		*)
		MesIDRack_UdcMin_Cell   		: WORD ; (* 	(NA) Min Cell Voltage String [CellVMinStr]      		*)
		MesIDModule_UdcMin_Cell 		: WORD ; (* 	(NA) Min Cell Voltage Module [CellVMinMod]      		*)
		MesIDCell_UdcMin		 		: WORD ; (* 	(NA) Max Cell Voltage [CellVMaxMod]      				*)	
		
		MesUdc_Cell						: WORD ; (*    (mV) Average cell voltage rack   						*)
	                                                                                                            
		// Rack			                                                                                        
																								                
		MesUdcMax_Rack          		: REAL ; (* 	(V) Max String Voltage [StrVMax]                		*)
		MesIDRack_UdcMax_Rack   		: WORD ; (* 	(NA) Max Cell Voltage String [StrVMaxStr]       		*)
		                                                                                                        
		MesUdcMin_Rack          		: REAL ; (* 	(V) Min Cell Voltage [StrVMin]                  		*)
		MesIDRack_UdcMin_Rack   		: WORD ; (* 	(NA) Min Cell Voltage String [StrVMinStr]       		*)
		                                                                                                        
		MesUdc_Rack						: REAL ; (* 	(V) Voltage of the cells, average [StrVAvg]				*)           	

	MesSystemOperationState			: WORD ;
	MesStatusConnectionProcess		: WORD ;
	MesSystemChargeState            : WORD ; (* 	         			*)                                 	                                                        	
	MesIDRack              	: WORD ; (* 	(NA) Battery Event 1 Bitfield [Evt1]             			*) 
	MesIDRackWState				: WORD ; (* 	                     			*)
	MesIDRackCriticalState          : WORD ; (* 	                   			*)  	
	MesBAUState				: WORD ;
                                                	                                                        	
	MesInsulation					: REAL ; (* 	(KΩ) 														*)      	

	AX_RACK							: ARRAY[1..CstNbRack_BAT_G] OF RackString_NARADA;
	AX_HVAC							: ARRAY[1..4] OF HVAC_NARADA ;
	
END_STRUCT
END_TYPE

// ---- 01_Equipement_Library/Batteries/BAT_SAMS.TcDUT
///////////
// Structure For Battery Controller. Main Operating Data to be saved ( ex: OPC ) .  
//////////

TYPE BAT_SAMS :
STRUCT
	
	MesData						: BAT ;   			(* MESA Data model *)

	AX_Rack						: ARRAY[1..CstNbRack_BAT_G] OF Rack_SAMS;	(* Object *)
	
	MesHeartBeat				: UINT;			(* (NA) Goes from 0 to 999 every s *)
	MesNbRackConnected			: UINT;			(* (NA) Nb of Racks in service ( strings ) *)
	MesNbRackTot				: UINT;			(* (NA) Total Nb of Racks (strings )*)
	MesIdcConnected				: REAL;			(* (A) Summation of all racks		*)
	MesUdcConnected				: REAL;			(* (V) Voltage connected ( average )*)
	MesUdcConnectedMedian		: REAL;			(* (V) Voltage connected ( median )*)
	MesUdcConnectedMax			: REAL;			(* (V) Voltage connected ( max )*)
	MesUdcConnectedMin			: REAL;			(* (V) Voltage connected ( min )	*)
	MesSoCConnected				: REAL; 		(* (%) SoC average ( priority : 1 if one is 0 all are 0, 2 : one is 100 all are 100, 3 : average )*)
	MesSoCConnectedMedian		: REAL; 		(* (%) SoC median value 	*)
	MesSoCConnectedMax			: REAL; 		(* (%) SoC Max value*)
	MesSoCConnectedMin			: REAL; 		(* (%) SoC Min value*)

	MesUdcMedian				: REAL;			(* (V) Voltage of the rack, median*)
	MesUdcMax					: REAL;			(* (V) Voltage of the rack, max*)
	MesUdcMin					: REAL;			(* (V) Voltage of the rack, min*)

	MesSoCMedian				: REAL; 		(* (%) SoC Median*)
	MesSoCMax					: REAL; 		(* (%) SoC Max*)
	MesSoCMin					: REAL; 		(* (%) SoC Min*)

	MesSoHMedian				: REAL; 		(* (%) SoH Median*)
	MesSoHMax					: REAL; 		(* (%) SoH Max*)
	MesSoHMin					: REAL; 		(* (%) SoH Min*)
	MesUdc_Cell					: REAL; 		(* (V)  Cell voltage among all strings in system. Average*)
	MesUdcMedian_Cell			: REAL; 		(* (V)  Cell voltage among all strings in system. Median*)
	MesUdcMax_Cell				: REAL; 		(* (V)Cell voltage among all strings in system. Max	*)
	MesUdcMax_Cell_RackID		: UINT:=1 ; 	(* (V)Rack ID where Cell voltage among all strings in system reaches Max value. *)
	MesUdcMin_Cell				: REAL; 		(* (V) Cell voltage among all strings in system. Min*)
	MesUdcMin_Cell_RackID		: UINT :=1 ; 	(* (V)Rack ID where Cell voltage among all strings in system reaches Min value. *)
	MesUdcDiffMax_Cell			: REAL; 		(* (V) Max Cell voltage difference among all strings in system. Min*)
	MesUdcDiffMax_Cell_RackID	: UINT:=1 ; 	(* (V)Rack ID where Cell voltage among all strings in system reaches Min value.*)
	MesTmp_Cell					: REAL; 		(* (°C)  Cell Temperature among all strings in system. Average*)
	MesTmpMedian_Cell			: REAL; 		(* (°C)  Cell Temperature among all strings in system. Median*)
	MesTmpMax_Cell				: REAL; 		(* (°C)Cell Temperature among all strings in system. Max*)
	MesTmpMax_Cell_RackID		: UINT:=1 ; 	(* (°C)Rack ID where Cell Temperature among all strings in system reaches Max value. *)
	MesTmpMin_Cell				: REAL; 		(* (°C) Cell Temperature among all strings in system. Min*)
	MesTmpMin_Cell_RackID		: UINT:=1 ; 	(* (°C)Rack ID where Cell Temperature among all strings in system reaches Min value. *)
	MesTmpDiffMax_Cell			: REAL; 		(* (°C) Max Cell Temperature difference among all strings in system. *)
	MesTmpDiffMax_Cell_RackID	: UINT:=1 ; 	(* (°C)Rack ID where Cell Temperature among all strings in system reaches Max diff value*)


	MesWatchdog					: WORD;			(* (NA) Inverses the WatchdogQuery	*)
	MesUdc_PartialOp			: REAL ; 		(* (V) Voltage of the Rack with the highest number of strings which are under Partial Op due to limit of voltage difference alarm*)
	MesUdc_PartialOp_RackID		: UINT:=1 ; 	(* (V) Rack ID where Voltage of the Rack with the highest number of strings which are under Partial Op due to limit of voltage difference alarm*)
	MesUdc_PartialOp_StringID	: UINT:=1 ; 	(* (V) Rack ID where Voltage of the Rack with the highest number of strings which are under Partial Op due to limit of voltage difference alarm*)
	MesSystemCommandStatus		: WORD ; 		(* Command status *)
	MesSystemMode				: WORD;			(* (NA) SystemMode read from the Battery*)
	MesSystemMode2				: WORD;			(* (NA) SystemMode2 read from the Battery*)
	
	MesDiStatus					: WORD;			(* (NA) DI Status*)
	MesDoStatus					: WORD;			(* (NA) DI Status*)
	MesSystemConfig1			: WORD ; 		(* Samsung State word Config 1*)
	MesSystemConfig2			: WORD ;    	(* Samsung State word Config 2*)
	MesRackStringState			: WORD ;    	(* Samsung State word Rack state*)

	ParamStringNbMin			: UINT ; 		(* Minimal number of strings Operable in order to works set at BBMS *)
	ParamUdiff					: REAL ;		(* Maximum voltage difference between  string for connexion set in BBMS . *)
	
// Evaluate	
	MesUdcMin_RackID			: UINT:=1 ;		(* (NA) Id of the Rack with the minimum Udc*)
	MesUdcMax_RackID			: UINT:=1 ;		(* (NA) Id of the Rack with the maximum Udc*)
	MesEconnected 				: REAL; 		(* Energy available for charge / discharge in the system BBMS. *)
	MesNbRackNormal				: UINT; 		(* Number of racks without alarms. *)

	                        	                
	MesAlarm1					: WORD;			(* (NA) Alarm1 read from the Battery System BMS*)
	MesAlarm2					: WORD;			(* (NA) Alarm2 read from the Battery System BMS*)
	MesRackAlarm1				: WORD;			(* (NA) Rack Alarm1 read from the Battery*)
	MesRackAlarm2				: WORD;			(* (NA) Rack Alarm2 read from the Battery*)
	MesRackProtection1			: WORD;			(* (NA) Rack Protection1 read from the Battery*)
	MesRackProtection2			: WORD;			(* (NA) Rack Protection2 read from the Battery*)
	MesRackStringAlarm1			: WORD;			(* (NA) Rack Alarm1 read from the Battery*)
	MesRackStringAlarm2			: WORD;			(* (NA) Rack Alarm2 read from the Battery*)
	MesRackStringAlarm3			: WORD;			(* (NA) Rack Alarm3 read from the Battery*)
	MesRackStringAlarm4			: WORD;			(* (NA) Rack Alarm4 read from the Battery*)		
	MesRackStringProtection1	: WORD;			(* (NA) Rack Protection1 read from the Battery*) 
	MesRackStringProtection2	: WORD;			(* (NA) Rack Protection2 read from the Battery*) 
	MesRackStringProtection3	: WORD;			(* (NA) Rack Protection3 read from the Battery*) 
	MesRackStringProtection4	: WORD;			(* (NA) Rack Protection4 read from the Battery*)	


	
	
END_STRUCT
END_TYPE

// ---- 01_Equipement_Library/Batteries/BAT_SAFT.TcDUT
///////////
// Structure For Battery Controller. Main Operating Data to be saved ( ex: OPC ) .  
//////////

TYPE BAT_SAFT :
STRUCT
	
	MesData						: BAT ;   			(* MESA Data model *)

	Rack						: ARRAY[1..CstNbRack_BAT_G] OF RackString_SAFT;	(* Object *)

	SubBMS						: ARRAY[1..1] OF BMS_SAFT ; 

	
	
	MesNbSubBMS				: WORD;		//(kWh) SubBank Count [NBSB]                   
	MesEToFullCharge        : REAL;		//(kWh) ToFullChargeEnergy [ToFullChargeEnergy]
	MesEconnected   		: REAL;		//(kWh) RemainingEnergy [RemainingEnergy]      
	MesP_Aux                : REAL;		//(kW) AUX Active Power [AUX ActPow]           
	MesS_Aux                : REAL;		//(kVA) AUX Apparent Power [AUX AppaPow]       
	MesQ_Aux                : REAL;		//(kVAr) AUX Reactive Power [AUX ReactPow]     
	MesEreact_Aux           : REAL;		//(kVArh) AUX   Cumulated   Reactive           
	MesEact_Aux             : REAL;		//Energy [AUX CumulReactEne]                   
	MesEapp_Aux             : REAL;		//"(kWh) AUX     Cumulated     Active          
	MesSoC_Uncertainty      : REAL;		//Energy [AUX CumulActEne]                     
	MesSoEMin               : REAL;		//(kVAh) AUX   Cumulated   Apparent            
	MesSoEMax               : REAL;		//Energy [AUX CumulAppaEne]                    


	MesUdcConnected				: REAL;			(* (V) Voltage connected ( average )*)	
	MesSoCConnected				: REAL; 		(* (%) SoC average ( priority : 1 if one is 0 all are 0, 2 : one is 100 all are 100, 3 : average )*)
	MesUdcMax					: REAL;			(* (V) Voltage of the rack, max*)
	MesUdcMin					: REAL;			(* (V) Voltage of the rack, min*)	
	MesNbRackConnected			: UINT;			(* (NA) Nb of Racks in service ( strings ) *)
	MesNbRackTot				: UINT;			(* (NA) Total Nb of Racks (strings )*)	
	
	
	
	
	
	
END_STRUCT
END_TYPE

// ---- 01_Equipement_Library/Batteries/BAT_Standard.TcDUT
{attribute 'pack_mode' := '1'}

TYPE BAT_Standard :
STRUCT
	AX_Rack						: ARRAY[1..CstNbRack_BAT_G] OF RACK;	(* Object *)
	
	MesData						: BAT;	(* Object *)	
	
END_STRUCT
END_TYPE

// ---- 01_Equipement_Library/Batteries/Module.TcDUT
///////////
// Structure For Battery Racks. Main Operating Data to be saved ( ex: OPC ) .  
//////////
TYPE Module :
STRUCT
	
	
	// Cell	: CELL ; 

// Model Module
MesID_String         :WORD;//(NA) STRING Index [StrIdx]                     
MesID_Module         :WORD;//(NA) Module Index [ModIdx]                     
MesNbCellTot         :WORD;//(NA) Module Cell Count [NCell]                 
                            
MesUdc               :REAL;//(NA) Module SoH [SoH]                          
MesUdcMax_Cell       :REAL;//(NA) Cycle Count [NCyc]                        
                                    
MesUdcMin_Cell       :REAL;//(V) Max Cell Voltage [CellVMax]                
MesIDCell_UdcMin_Cell:WORD;//(NA) Max Cell Voltage Cell [CellVMaxCell]      
MesUdc_Cell          :REAL;//(V) Min Cell Voltage [CellVMin]                
MesTempMax_Cell      :REAL;//(NA) Min Cell Voltage Cell [CellVMinCell]      
                         
MesTempMin_Cell      :REAL;//(C) Max Cell Temperature [CellTmpMax]          
                          
MesTemp_Cell         :REAL;//(C) Min Cell Temperature [CellTmpMin]          
MesNbCellBalancing   :WORD;//(NA) Min Cell Temperature Cell [CellTmpMinCell]
MesID_SerialNb		 :WORD;//(C) Average Cell Temperature [CellTmpAvg]      





// Model String			
MesNbCell				: WORD;//(NA) Module Cell Count [ModNCell]                 
MesSoC                  : REAL;//(NA) Module SoC [ModSoC]                          
MesSoH                  : REAL;//(NA) Module SoH [ModSoH]                          
//MesUdcMax_Cell        : REAL;//(V) Max Cell Voltage [ModCellVMax]                
MesIDCell_UdcMax_Cell   : REAL;//(NA) Max Cell Voltage Cell [ModCellVMaxCell]      
//MesUdcMin_Cell          : REAL;//(V) Min Cell Voltage [ModCellVMin]                
//MesIDCell_UdcMin_Cell   : WORD;//(NA) Min Cell Voltage Cell [ModCellVMinCell]      
//MesUdc_Cell             : REAL;//(V) Average Cell Voltage [ModCellVAvg]            
//MesTempMax_Cell         : REAL;//(C) Max Cell Temperature [ModCellTmpMax]          
MesIDCell_TempMax_Cell  : REAL;//(NA) Max Cell Temperature Cell [ModCellTmpMaxCell]
//MesTempMin_Cell         : REAL;//(C) Min Cell Temperature [ModCellTmpMin]          
MesIDCell_TempMin_Cell  : REAL;//(NA) Min Cell Temperature Cell [ModCellTmpMinCell]
//MesTemp_Cell			: REAL;//(C) Average Cell Temperature [ModCellTmpAvg]      



 















































END_STRUCT
END_TYPE

// ---- 01_Equipement_Library/Batteries/CELL.TcDUT
///////////
// Structure For Battery Racks. Main Operating Data to be saved ( ex: OPC ) .  
//////////
TYPE CELL :
STRUCT
	
	




END_STRUCT
END_TYPE

// ---- 01_Equipement_Library/Batteries/BMS_SAFT.TcDUT
///////////
// Structure For Battery Racks. Main Operating Data to be saved ( ex: OPC ) .  
//////////
TYPE BMS_SAFT :
STRUCT
	
HVAC 				: HVAC_SAFT ;	


MesEToFullCharge				: REAL   ;//(kWh) ToFullChargeEnergy [SubBankToFullChargeEnergy]             
MesEconnected                   : REAL   ;//(kWh) RemainingEnergy [SubBankRemainingEnergy]                   
//HVAC.MesTempExt                 : REAL   ;//(C) HVAC Outside Temp [SubBankHVACOutTemp]                       
//HVAC.MesTemp                    : REAL   ;//(C) HVAC Inside Temp [SubBankHVACInTemp]                         
//HVAC.MesHygro                   : REAL   ;//(%) HVAC Inside Humidity [SubBankInsideHumidity]                 
//                                : REAL   ;//(NA) SetPointInsideTemperature [SubBankSetPointInsideTemperature]
//                                : REAL   ;//(NA) SetPointInsideHumidity [SubBankSetPointInsideHumidity]      
MesU_Aux                        : REAL   ;//(NA) AUX Average Line Voltage [SubBankAUX Avg Volt]              
MesFreq_Aux                     : REAL   ;//(NA) AUX Frequency [SubBankAUX Freq]                             
MesP_Aux                        : REAL   ;//(kW) AUX Active Power [SubBankAUX ActPow]                        
MesS_Aux                        : REAL   ;//(kVA) AUX Apparent Power [SubBankAUX AppaPow]                    
MesQ_Aux                        : REAL   ;//(kVAr) AUX Reactive Power [SubBankAUX ReactPow]                  
MesEreact_Aux        : REAL   ;//(kVArh) AUX   Cumulated   Reactive                               
MesEact_Aux          : REAL   ;//Energy [SubBankAUX CumulReactEne]                                
MesEapp_Aux          : REAL   ;//(kWh) AUX     Cumulated     Active                               
//HVAC.MesIDState                 : WORD   ;//Energy [SubBankAUX CumulActEne]                                  
MesIDAlarm                      : WORD   ;//(kVAh) AUX   Cumulated   Apparent                                
MesIDAlarm2                     : WORD   ;//Energy [SubBankAUX CumulAppaEne]                                 



































END_STRUCT
END_TYPE

// ---- 01_Equipement_Library/Batteries/Rack.TcDUT
{attribute 'pack_mode' := '1'}

TYPE Rack :
STRUCT
	
		// Info of Rack BBMS  
		ParamNbStrings			: UINT ; 	// 		Number of strings for the rack set in BBMS 
		MesHeartBeat			: UINT;		// (NA) Rack's Heartbeat, increases by 1 every second
		MesAlarm1				: WORD;		// (NA) bit0: 
		MesAlarm2				: WORD;		// (NA) bit0: 
		MesProtection1			: WORD;		// (NA) bit0: 
		MesProtection2			: WORD;		// (NA) bit0: 		
		MesSwitchControlStatus	: WORD ; 	// Control status
		MesSwitchSensorStatus	: WORD ; 	// Sensor status
		MesUSwtchGrPackPlus		: REAL;		// (V)	a measured value of voltage applied to pack(+) of switchgear
		MesTempPCB				: REAL ; 	// (°C) Temperature Rack PCB 
		MesIdcFaultLvl			: UINT ;	//		Current Level when power is cut (1/2/3/4/5/6/7/8/9/10 : 1200A/700A/500A/200A/0A/-0A/-200A/-500A/-700A/-1200A)
		MesDcOpenCount			: UINT ; 	// Count number of dc opening 
		MesDcCloseCount			: UINT ; 	// Count number of dc closing 
		
		AX_RACKSTRING			: ARRAY[1..1] OF RackString ; 	// object 
	
		CalRackClosed			: BOOL ; 		// Rack ( Main DC contactor )is closed 

END_STRUCT
END_TYPE

// ---- 01_Equipement_Library/Batteries/RackString_NARADA.TcDUT
///////////
// Structure For Battery Racks. Main Operating Data to be saved ( ex: OPC ) .  
//////////
TYPE RackString_NARADA :
STRUCT
	
		MesData		: RackString ;
	
		MesIDWarning						: WORD;
		MesIDCriticalAlarm					: WORD;		
 
		MesInsulationValue          		: REAL  ; (* (Ω) 	*)
		MesPositiveInsulationValue          : REAL  ; (* (Ω)  	*)    
		MesNegativeInsulationValue          : REAL  ; (* (Ω)  	*)            	
	                                                     
		MesCCL						        : REAL  ; (* (A)  	*)     
		MesDCL						        : REAL  ; (* (A)  	*)  

		MesIDstate2				 			: REAL  ; (* Rack Charge State (Chg/Dsg) - 0x0: (Idle); 0x1: (Discharging); 0x2: Charging) *)
		
		MesNaradaIDState					: UINT ;  (* 	0 : Normal ;  1 : Interdit la charge ; 2 : Interdire la décharge ; 3 : Standby ; 4 : Arrêt *)
		
END_STRUCT
END_TYPE

// ---- 01_Equipement_Library/Batteries/RackString_SAFT.TcDUT
///////////
// Structure For Battery Racks. Main Operating Data to be saved ( ex: OPC ) .  
//////////
TYPE RackString_SAFT :
STRUCT
	
		MesData		: RackString ;
		Module		: ARRAY[1..CstNbModule_Rack_G] OF  Module ; 
		
     	
	
		

		
		
		
		
		
		
		
	
END_STRUCT
END_TYPE

// ---- 01_Equipement_Library/Batteries/RackString.TcDUT
///////////
// Structure For Battery Racks. Main Operating Data to be saved ( ex: OPC ) .  
//////////
TYPE RackString :
STRUCT
	
//Model Li Ion
MesNbModuleTot				: WORD  ; //(NA) Module Count [StrNMod]                         
MesIDState                  : DWORD  ; //(NA) String Status [StrSt]                          
MesIDConnectAlarm           : UINT  ; //(NA) Connection Failure Reason [StrConFail]         
MesSoC                      : REAL  ; //(%) String State of Charge [StrSoC]                 
MesSoH                      : REAL  ; //(%) String State of Health [StrSoH]                 
MesIdc                      : REAL  ; //(A) String Current [StrA]                            
MesUdc                      : REAL  ; //(V) String Voltage [V]                           
MesUdcMax_Cell              : REAL  ; //(V) Max Cell Voltage [StrCellVMax]                  
MesIDModule_UdcMax_Cell     : WORD  ; //(NA) Max Cell Voltage Module [StrCellVMaxMod]       
MesUdcMin_Cell              : REAL  ; //(V) Min Cell Voltage [StrCellVMin]                  
MesIDModule_UdcMin_Cell     : WORD  ; //(NA) Min Cell Voltage Module [StrCellVMinMod]       
MesUdc_Cell                 : REAL  ; //(V) Average Cell Voltage [StrCellVAvg]              
MesTempMax_Module           : REAL  ; //(C) Max Module Temperature [StrModTmpMax]           
MesIDModule_TempMax_Module  : WORD  ; //(NA) Max Module Temperature Module [StrModTmpMaxMod]
MesTempMin_Module           : REAL  ; //(C) Min Module Temperature [StrModTmpMin]           
MesIDModule_TempMin_Module  : WORD  ; //(NA) Min Module Temperature Module [StrModTmpMinMod]
MesTemp_Module              : REAL  ; //(C) Average Module Temperature [StrModTmpAvg]       
MesIDDisableReason          : WORD  ; //(NA) Disabled Reason [StrDisRsn]                    
MesIDState_DCSwitch         : WORD  ; //(NA) Contactor Status [StrConSt]                    
MesIDAlarm                  : DWORD  ; //(NA) String Event 1 [StrEvt1]     

MesIDAlarm_Vendor1          : DWORD  ;//(NA) Vendor Event Bitfield 1 [StrEvtVnd1]           
     
MesSoC_Uncertainty			: REAL  ;//(%) SOC Uncertainty [SOC Uncertainty]       

MesID_String				:WORD  ;//(NA) STRING Index [Idx]                          	
MesNbCellbalancing          :WORD  ;//(NA) String Cell Balancing Count [NCellBal]      
MesDoD                      :REAL  ;//(%) String Depth of Discharge [DoD]         

END_STRUCT
END_TYPE

// ---- 01_Equipement_Library/Batteries/RackString_KP.TcDUT
///////////
// Structure For Battery Racks. Main Operating Data to be saved ( ex: OPC ) .  
//////////
TYPE RackString_KP :
STRUCT
	
		MesData		: RackString ;

		
     	
	
		

		
		
		
		
		
		
		
	
END_STRUCT
END_TYPE

// ---- 01_Equipement_Library/Batteries/Rack_SAMS.TcDUT
///////////
// Structure For Battery Racks. Main Operating Data to be saved ( ex: OPC ) .  
//////////
TYPE Rack_SAMS :
STRUCT
	
		// Info of Rack BBMS  
	
		MesData					: Rack ; 
		
		ParamNbStrings			: UINT ; 	// 		Number of strings for the rack set in BBMS 
		MesHeartBeat			: UINT;		// (NA) Rack's Heartbeat, increases by 1 every second
		MesAlarm1				: WORD;		// (NA) bit0: 
		MesAlarm2				: WORD;		// (NA) bit0: 
		MesProtection1			: WORD;		// (NA) bit0: 
		MesProtection2			: WORD;		// (NA) bit0: 		
		MesSwitchControlStatus	: WORD ; 	// Control status
		MesSwitchSensorStatus	: WORD ; 	// Sensor status
		MesUSwtchGrPackPlus		: REAL;		// (V)	a measured value of voltage applied to pack(+) of switchgear
		MesTempPCB				: REAL ; 	// (°C) Temperature Rack PCB 
		MesIdcFaultLvl			: UINT ;	//		Current Level when power is cut (1/2/3/4/5/6/7/8/9/10 : 1200A/700A/500A/200A/0A/-0A/-200A/-500A/-700A/-1200A)
		MesDcOpenCount			: UINT ; 	// Count number of dc opening 
		MesDcCloseCount			: UINT ; 	// Count number of dc closing 
		
		AX_RACKSTRING			: ARRAY[1..1] OF RackString_SAMS ; 	// object 
	
		CalRackClosed			: BOOL ; 		// Rack ( Main DC contactor )is closed 

END_STRUCT
END_TYPE

// ---- 01_Equipement_Library/Batteries/RackString_SAMS.TcDUT
///////////
// Structure For Battery Racks. Main Operating Data to be saved ( ex: OPC ) .  
//////////
TYPE RackString_SAMS :
STRUCT
		MesData		: RackString ;
	
		MesMode								: UINT;		// (NA) Rack mode: 0: None, 1: Init, 2: Off, DcSwitch On, 3: On, DcSwitch On,
		MesAlarm1							: WORD;		// (NA) bit0: 
		MesAlarm2							: WORD;		// (NA) bit0: 
		MesAlarm3							: WORD;		// (NA) bit0: 
		MesAlarm4							: WORD;		// (NA) bit0: 
		MesProtection1						: WORD;		// (NA) bit0: 
		MesProtection2						: WORD;		// (NA) bit0: 
		MesProtection3						: WORD;		// (NA) bit0: 
		MesProtection4						: WORD;		// (NA) bit0: 		
		MesControlStatus					: WORD ; 	// Control Status
		
		MesUdc_ModuleSum					: REAL  ;	// String voltage obtained by summing module voltage 
		MesUdc_CellSum						: REAL ; 	// String voltage obtained by summing Cell voltage 
	
		MesIdc_Avg							: REAL;		// (A) Rack Current ( average of 3 sec) 

		MesCCL								: REAL;		// (A) Charge limit of rack
		MesDCL								: REAL;		// (A) Discharge limit of rack
		MesCPL								: REAL ; 	// (kW) Charge Power Limit		- To zero if Estop is set . 
		MesDPL								: REAL ; 	// (kW) Discharge Power Limit - To zero if Estop is set .
		MesECharge							: REAL ; 	// (kWh) Total Energy charged over time 
		MesEDischarge						: REAL ; 	// (kWh) Total Energy Discharge over time 
		MesOff_ModuleID						: UINT; 	// Module ID where the power is off while the other modules are connected . 
		MesComError_ModuleID				: UINT ; 	// Module ID where there is a LOC while other modules are connected . 
		MesUdcDiffMax_Cell					: REAL ; 	// (V) 	Max voltage difference between cells . 
		
		
		MesUdcMax1_Cell_CellID				: UINT; 	// (V)	Cell ID where Cell voltage reaches Max value. Rank #1
		
		MesUdcMin1_Cell_CellID				: UINT; 	// (V)	Cell ID where Cell voltage reaches Min value. Rank #1
		MesUdcMax2_Cell						: REAL; 	// (V)	Cell voltage . Max Rank #2
		MesUdcMax2_Cell_ModuleID			: UINT; 	// (V)	Module ID where Cell voltage  reaches Max value. Rank #2
		MesUdcMax2_Cell_CellID				: UINT; 	// (V)	Cell ID where Cell voltage reaches Max value. Rank #2
		MesUdcMin2_Cell						: REAL; 	// (V)	Cell voltage . Min Rank #2
		MesUdcMin2_Cell_ModuleID			: UINT; 	// (V)	Module ID where Cell voltage  reaches Min value. Rank #2
		MesUdcMin2_Cell_CellID				: UINT; 	// (V)	Cell ID where Cell voltage reaches Min value. Rank #2		
		MesTempDiffMax_Cell					: REAL ; 	// (°C) Max Temp difference between cells . 
		MesTemp_Cell						: REAL; 	// (°C)	Cell Temp . Average
		MesTempMax1_Cell					: REAL; 	// (°C)	Cell Temp . Max Rank #1
		MesTempMax1_Cell_ModuleID			: UINT; 	// (°C)	Module ID where Cell Temp  reaches Max value. Rank #1
		MesTempMax1_Cell_CellID				: UINT; 	// (°C)	Cell ID where Cell Temp reaches Max value. Rank #1
		MesTempMin1_Cell					: REAL; 	// (°C)	Cell Temp . Min Rank #1
		MesTempMin1_Cell_ModuleID			: UINT; 	// (°C)	Module ID where Cell Temp  reaches Min value. Rank #1
		MesTempMin1_Cell_CellID				: UINT; 	// (°C)	Cell ID where Cell Temp reaches Min value. Rank #1
		MesTempMax2_Cell					: REAL; 	// (°C)	Cell Temp . Max Rank #2
		MesTempMax2_Cell_ModuleID			: UINT; 	// (°C)	Module ID where Cell Temp  reaches Max value. Rank #2
		MesTempMax2_Cell_CellID				: UINT; 	// (°C)	Cell ID where Cell Temp reaches Max value. Rank #2
		MesTempMin2_Cell					: REAL; 	// (°C)	Cell Temp . Min Rank #2
		MesTempMin2_Cell_ModuleID			: UINT; 	// (°C)	Module ID where Cell Temp  reaches Min value. Rank #2
		MesTempMin2_Cell_CellID				: UINT; 	// (°C)	Cell ID where Cell Temp reaches Min value. Rank #2		
		MesTempPCBMax						: REAL ; 	// (°C) Temperature PCB Max
		MesTempPCBMax_ModuleID				: UINT ;    // (°C) Temperature PCB Max module ID
		MesTempPCBMin						: REAL ;    // (°C) Temperature PCB Min
		MesTempPCBMin_ModuleID				: UINT ; 	// (°C) Temperature PCB Min Module ID 	
		MesSensorStatus						: UINT ; 	//	Register status (only for Samsung diagnosis)
		MesModuleScanStatus					: UINT ; 	//	Register status (only for Samsung diagnosis)
		MesModuleBalancingStatus			: UINT ; 	//	Register status (only for Samsung diagnosis)
		MesModuleAddressStatus				: UINT ; 	//	Register status (only for Samsung diagnosis)
		MesModuleVoltageStatus				: UINT ; 	//	Register status (only for Samsung diagnosis)	
		MesModuleTemperatureStatus			: UINT ; 	//	Register status (only for Samsung diagnosis)
		MesUdcDiffCellMax					: REAL ; 	// (V)[Rack#1][String#1] Difference Voltage (MAX(Cell Sensing Summation))
		MesUdcDiffModuleMax					: REAL ; 	// (V)[Rack#1][String#1] Difference Voltage (Max(Module Sensing))        
		MesUdcDiffModuleMax_ModuleID		: UINT ; 	// [Rack#1][String#1] Difference Voltage (Max) Module Position           
		MesUdcDiffCellMin					: REAL ; 	// (V)[Rack#1][String#1] Difference Voltage (Min(Cell Sensing Summation))
		MesUdcDiffModuleMin					: REAL ; 	// (V)[Rack#1][String#1] Difference Voltage (Min(Module Sensing))        
		MesUdcDiffModuleMin_ModuleID		: UINT ; 	// [Rack#1][String#1] Difference Voltage (Min) Module Position           
//		MesState							: UINT ; 	// internal string state machine . 
		MesCellVDist_under20mV				: REAL ; 	// (%)[Rack#1][String#1] Cell V Distribution (Under 20mV)
		MesCellVDist_underVimbAlarm 		: REAL ; 	// (%)[Rack#1][String#1] Cell V Distribution (Under V-IMB Alarm Level)
		MesCellVDist_underVimbProtection 	: REAL ; 	// (%)[Rack#1][String#1] Cell V Distribution (Under V-IMB Protection Level)
		MesCellVDist_VimbProtection 		: REAL ; 	// (%)[Rack#1][String#1] Cell V Distribution (V-IMB Protection Level or More)
		MesCellBalancingCntMax				: UINT ; 	// ()[Rack#1][String#1] Cell Balancing Execution Count (Max)
		MesCellBalancingCntMax_ModuleID		: UINT ; 	// ()[Rack#1][String#1] Cell Balancing Execution Count (Max) Module Position
		MesCellBalancingCntMax_CellID		: UINT ; 	// ()[Rack#1][String#1] Cell Balancing Execution Count (Max) Cell Position
		MesMaxBalancingTime					: REAL ; 	// (min)[Rack#1][String#1] Max Balancing Time (minute)
		
	
END_STRUCT
END_TYPE

// ---- 01_Equipement_Library/Batteries/St_AlarmCodeSamsung.TcDUT
TYPE St_AlarmCodeSamsung :
STRUCT
	

// System Alarm1 bAlarm1	
BMS_Protection4_module_pcb_ut              : BOOL; 		// SystemBms Protection 4 : module pcb ut
BMS_Protection4_module_pcb_ot              : BOOL; 		// SystemBms Protection 4 : module pcb ot
BMS_Protection4_dcsw_count_fail            : BOOL; 		// SystemBms Protection 4 : dcsw count fail
                                           				// 
                                           				// 
                                           				// 
                                           				// 
                                           				// 
BMS_Protection4_fuse_or_dcsw_sensing_fail  : BOOL; 		// SystemBms Protection 4 : fuse or dcsw sensing fail
                                           				// 
                                           				// 
                                           				// 
                                           				// 
                                           				// 
                                           				// 
                                           				// 
														// : wAlarmCode



// System Alarm1 bAlarm1
                                           				// 
                                           				// 
                                           				// 
                                           				// 
                                           				// 
                                           				// 
                                           				// 
                                           				// 
BMS_Protection3_dcsw1_sensing_fail         : BOOL; 		// SystemBms Protection3 : dcsw1_sensing_fail
BMS_Protection3_dcsw2_sensing_fail         : BOOL; 		// SystemBms Protection3 : dcsw2_sensing_fail
BMS_Protection3_dcsw1_fail                 : BOOL; 		// SystemBms Protection3 : dcsw1_fail
BMS_Protection3_dcsw2_fail                 : BOOL; 		// SystemBms Protection3 : dcsw2_fail
BMS_Protection3_fan_fail_Option            : BOOL; 		// SystemBms Protection3 : fan fail [Option]
BMS_Protection3_additional_protection_fail : BOOL; 		// SystemBms Protection3 : additional protection fail
BMS_Protection3_cell_chg_operation_limit   : BOOL; 		// SystemBms Protection3 : cell chg operation limit
BMS_Protection3_cell_dchg_operation_limit  : BOOL; 		// SystemBms Protection3 : cell dchg operation limit
														// : wAlarmCode



// System Alarm1 bAlarm1
BMS_Protection1_module_UT                  : BOOL; 		// SystemBms Protection1 : module UT
BMS_Protection1_module_OT                  : BOOL; 		// SystemBms Protection1 : module OT
BMS_Protection1_module_UV                  : BOOL; 		// SystemBms Protection1 : module UV
BMS_Protection1_module_OV                  : BOOL; 		// SystemBms Protection1 : module OV
BMS_Protection1_module_V_imb               : BOOL; 		// SystemBms Protection1 : module V-imb
BMS_Protection1_module_T_imb               : BOOL; 		// SystemBms Protection1 : module T-imb
BMS_Protection1_R_M_comm_fail              : BOOL; 		// SystemBms Protection1 : R-M comm fail
BMS_Protection1_R_S_comm_fail              : BOOL; 		// SystemBms Protection1 : R-S comm fail
BMS_Protection1_rack_ChgOC                 : BOOL; 		// SystemBms Protection1 : rack ChgOC
BMS_Protection1_rack_DchgOC                : BOOL; 		// SystemBms Protection1 : rack DchgOC
BMS_Protection1_rack_UV                    : BOOL; 		// SystemBms Protection1 : rack UV
BMS_Protection1_rack_OV                    : BOOL; 		// SystemBms Protection1 : rack OV
BMS_Protection1_rack_V_sensing_diff        : BOOL; 		// SystemBms Protection1 : rack V sensing diff
BMS_Protection1_rack_I_senser_fail         : BOOL; 		// SystemBms Protection1 : rack I senser fail
BMS_Protection1_rack_fuse_fail_Option      : BOOL; 		// SystemBms Protection1 : rack fuse fail [Option]
BMS_Protection1_permanent_uv               : BOOL; 		// SystemBms Protection1 : permanent  uv
														// : wAlarmCode



// System Alarm1 bAlarm1
BMS_Alarm4_module_pcb_ut                   : BOOL; 		// SystemBms Alarm4 : module pcb ut
BMS_Alarm4_module_pcb_ot                   : BOOL; 		// SystemBms Alarm4 : module pcb ot
BMS_Alarm4_dcsw_count_fail                 : BOOL; 		// SystemBms Alarm4 : dcsw count fail
                                           				//  
                                           				//  
                                           				//  
                                           				//  
                                           				//  
BMS_Alarm4_fuse_or_dcsw_sensing_fail       : BOOL; 		// SystemBmsAlarm4 : fuse or dcsw sensing fail
BMS_Alarm4_Rest_Cell_Balancing             : BOOL; 		// SystemBmsAlarm4 : Rest Cell Balancing
                                           				// 
                                           				// 
                                           				// 
                                           				// 
                                           				// 
                                           				// 
														// : wAlarmCode



// System Alarm1 bAlarm1
                                           				// 
                                           				// 
                                           				// 
                                           				// 
                                           				// 
                                           				// 
                                           				// 
                                           				// 
BMS_Alarm3_dcsw1_sensing_fail              : BOOL; 		// SystemBms Alarm3 : dcsw1_sensing_fail
BMS_Alarm3_dcsw2_sensing_fail              : BOOL; 		// SystemBms Alarm3 : dcsw2_sensing_fail
BMS_Alarm3_dcsw1_fail                      : BOOL; 		// SystemBms Alarm3 : dcsw1_fail
BMS_Alarm3_dcsw2_fail                      : BOOL; 		// SystemBms Alarm3 : dcsw2_fail
BMS_Alarm3_fan_fail_Option                 : BOOL; 		// SystemBms Alarm3 : fan fail [Option]
BMS_Alarm3_additional_protection_fail      : BOOL; 		// SystemBms Alarm3 : additional protection fail
BMS_Alarm3_cell_chg_operation_limit        : BOOL; 		// SystemBms Alarm3 : cell chg operation limit
BMS_Alarm3_cell_dchg_operation_limit       : BOOL; 		// SystemBms Alarm3 : cell dchg operation limit
														// : wAlarmCode





// System Alarm1 bAlarm1
BMS_Alarm1_module_UT                       : BOOL; 		//SystemBms Alarm1 : module UT
BMS_Alarm1_module_OT                       : BOOL; 		//SystemBms Alarm1 : module OT
BMS_Alarm1_module_UV                       : BOOL; 		//SystemBms Alarm1 : module UV
BMS_Alarm1_module_OV                       : BOOL; 		//SystemBms Alarm1 : module OV
BMS_Alarm1_module_V_imb                    : BOOL; 		//SystemBms Alarm1 : module V-imb
BMS_Alarm1_module_T_imb                    : BOOL; 		//SystemBms Alarm1 : module T-imb
BMS_Alarm1_R_M_comm_fail                   : BOOL; 		//SystemBms Alarm1 : R-M comm fail
BMS_Alarm1_R_S_comm_fail                   : BOOL; 		//SystemBms Alarm1 : R-S comm fail
BMS_Alarm1_rack_ChgOC                      : BOOL; 		//SystemBms Alarm1 : rack ChgOC
BMS_Alarm1_rack_DchgOC                     : BOOL; 		//SystemBms Alarm1 : rack DchgOC
BMS_Alarm1_rack_UV                         : BOOL; 		//SystemBms Alarm1 : rack UV
BMS_Alarm1_rack_OV                         : BOOL; 		//SystemBms Alarm1 : rack OV
BMS_Alarm1_rack_V_sensing_diff             : BOOL; 		//SystemBms Alarm1 : rack V sensing diff
BMS_Alarm1_rack_I_senser_fail              : BOOL; 		//SystemBms Alarm1 : rack I senser fail
BMS_Alarm1_rack_fuse_fail_Option           : BOOL; 		//SystemBms Alarm1 : rack fuse fail [Option]
BMS_Alarm1_permanent_uv                    : BOOL; 		//SystemBms Alarm1 : permanent  uv
														// : wAlarmCode



// System Alarm1 bAlarm1
Rack_Protection4_module_pcb_ut             : BOOL; 		//Rack Protection4 : module pcb ut
Rack_Protection4_module_pcb_ot             : BOOL; 		//Rack Protection4 : module pcb ot
Rack_Protection4_dcsw_count_fail           : BOOL; 		//Rack Protection4 : dcsw count fail
                                           				// 
                                           				// 
                                           				// 
                                           				// 
                                           				// 
Rack_Protection4_fuse_or_dcsw_sensing_fail : BOOL; 		//Rack Protection 4 : fuse or dcsw sensing fail
                                           				// 
                                           				// 
                                           				// 
                                           				// 
                                           				// 
                                           				// 
                                           				// 
														// : wAlarmCode


// System Alarm1 bAlarm1

                                          				// 
                                          				// 
                                          				// 
                                          				// 
                                          				// 
                                          				// 
                                          				// 
                                          				// 
Rack_Protection3_dcsw1_sensing_fail        : BOOL; 		//Rack Protection3 : dcsw1_sensing_fail
Rack_Protection3_dcsw2_sensing_fail        : BOOL; 		//Rack Protection3 : dcsw2_sensing_fail
Rack_Protection3_dcsw1_fail                : BOOL; 		//Rack Protection3 : dcsw1_fail
Rack_Protection3_dcsw2_fail                : BOOL; 		//Rack Protection3 : dcsw2_fail
Rack_Protection3_fan_fail_Option           : BOOL; 		//Rack Protection3 : fan fail [Option]
Rack_Protection3_additional_protection_fail: BOOL; 		//Rack Protection3 : additional protection fail
Rack_Protection3_cell_chg_operation_limit  : BOOL; 		//Rack Protection3 : cell chg operation limit
Rack_Protection3_cell_dchg_operation_limit : BOOL; 		//Rack Protection3 : cell dchg operation limit
														// : wAlarmCode





// System Alarm1 bAlarm1
Rack_Protection1_module_UT                 : BOOL; 		//Rack Protection1 : module UT
Rack_Protection1_module_OT                 : BOOL; 		//Rack Protection1 : module OT
Rack_Protection1_module_UV                 : BOOL; 		//Rack Protection1 : module UV
Rack_Protection1_module_OV                 : BOOL; 		//Rack Protection1 : module OV
Rack_Protection1_module_Vimb               : BOOL; 		//Rack Protection1 : module V-imb
Rack_Protection1_module_Timb               : BOOL; 		//Rack Protection1 : module T-imb
Rack_Protection1_RM_comm_fail              : BOOL; 		//Rack Protection1 : R-M comm fail
Rack_Protection1_RS_comm_fail              : BOOL; 		//Rack Protection1 : R-S comm fail
Rack_Protection1_rack_ChgOC                : BOOL; 		//Rack Protection1 : rack ChgOC
Rack_Protection1_rack_DchgOC               : BOOL; 		//Rack Protection1 : rack DchgOC
Rack_Protection1_rack_UV                   : BOOL; 		//Rack Protection1 : rack UV
Rack_Protection1_rack_OV                   : BOOL; 		//Rack Protection1 : rack OV
Rack_Protection1_rack_V_sensing_diff       : BOOL; 		//Rack Protection1 : rack V sensing diff
Rack_Protection1_rack_I_senser_fail        : BOOL; 		//Rack Protection1 : rack I senser fail
Rack_Protection1_rack_fuse_fail_Option     : BOOL; 		//Rack Protection1 : rack fuse fail [Option]
Rack_Protection1_permanent_uv              : BOOL; 		//Rack Protection1 : permanent  uv
														// : wAlarmCode



// System Alarm1 bAlarm1
Rack_Alarm4_module_pcb_ut                  : BOOL; 		//Rack Alarm4 : module pcb ut
Rack_Alarm4_module_pcb_ot                  : BOOL; 		//Rack Alarm4 : module pcb ot
Rack_Alarm4_dcsw_count_fail                : BOOL; 		//Rack Alarm4 : dcsw count fail
                                           				// 
                                           				// 
                                           				// 
                                           				// 
                                           				// 
Rack_Alarm4_fuse_or_dcsw_sensing_fail      : BOOL; 		//Rack Alarm4 : fuse or dcsw sensing fail
Rack_Alarm4_Rest_Cell_Balancing            : BOOL; 		//Rack Alarm4 : Rest Cell Balancing
                                           				// 
                                           				// 
                                           				// 
                                           				// 
                                           				// 
                                           				// 
														// : wAlarmCode

// System Alarm1 bAlarm1                                           				
                                           				// 
                                           				// 
                                           				// 
                                           				// 
                                           				// 
                                           				// 
                                           				// 
                                           				// 
Rack_Alarm3_dcsw1_sensing_fail             : BOOL; 		//Rack Alarm3 : dcsw1_sensing_fail
Rack_Alarm3_dcsw2_sensing_fail             : BOOL; 		//Rack Alarm3 : dcsw2_sensing_fail
Rack_Alarm3_dcsw1_fail                     : BOOL; 		//Rack Alarm3 : dcsw1_fail
Rack_Alarm3_dcsw2_fail                     : BOOL; 		//Rack Alarm3 : dcsw2_fail
Rack_Alarm3_fan_fail_Option                : BOOL; 		//Rack Alarm3 : fan fail [Option]
Rack_Alarm3_additional_protection_fail     : BOOL; 		//Rack Alarm3 : additional protection fail
Rack_Alarm3_cell_chg_operation_limit       : BOOL; 		//Rack Alarm3 : cell chg operation limit
Rack_Alarm3_cell_dchg_operation_limit      : BOOL; 		//Rack Alarm3 : cell dchg operation limit
														// : wAlarmCode


// System Alarm1 bAlarm1                                                   	
                                           				// 
                                           				// 
                                           				// 
                                           				// 
                                           				// 
                                           				// 
                                           				// 
                                           				// 
                                           				// 
                                           				// 
                                           				// 
                                           				// 
                                           				// 
                                           				// 
                                           				// 
                                           				// 
														// : wAlarmCode

// System Alarm1 bAlarm1                                                   	
Rack_Alarm1_module_UT                      : BOOL; 		//Rack Alarm1 : module UT
Rack_Alarm1_module_OT                      : BOOL; 		//Rack Alarm1 : module OT
Rack_Alarm1_module_UV                      : BOOL; 		//Rack Alarm1 : module UV
Rack_Alarm1_module_OV                      : BOOL; 		//Rack Alarm1 : module OV
Rack_Alarm1_module_Vimb                    : BOOL; 		//Rack Alarm1 : module V-imb
Rack_Alarm1_module_Timb                    : BOOL; 		//Rack Alarm1 : module T-imb
Rack_Alarm1_RM_comm_fail                   : BOOL; 		//Rack Alarm1 : R-M comm fail
Rack_Alarm1_RS_comm_fail                   : BOOL; 		//Rack Alarm1 : R-S comm fail
Rack_Alarm1_rack_ChgOC                     : BOOL; 		//Rack Alarm1 : rack ChgOC
Rack_Alarm1_rack_DchgOC                    : BOOL; 		//Rack Alarm1 : rack DchgOC
Rack_Alarm1_rack_UV                        : BOOL; 		//Rack Alarm1 : rack UV
Rack_Alarm1_rack_OV                        : BOOL; 		//Rack Alarm1 : rack OV
Rack_Alarm1_rack_V_sensing_diff            : BOOL; 		//Rack Alarm1 : rack V sensing diff
Rack_Alarm1_rack_I_senser_fail             : BOOL; 		//Rack Alarm1 : rack I senser fail
Rack_Alarm1_rack_fuse_fail_Option          : BOOL; 		//Rack Alarm1 : rack fuse fail [Option]
Rack_Alarm1_permanent_uv                   : BOOL; 		//Rack Alarm1 : permanent  uv
														// : wAlarmCode

END_STRUCT
END_TYPE

// ---- 01_Equipement_Library/Datalogger/Datalogger.TcDUT
TYPE Datalogger :
STRUCT
	MesAlarmCom					: BOOL ; 						(* (NA) Communication alarm *)
	MesAlarmCode				: WORD ; 						(* (NA) Internal Akuo Alarm Code				*)
	MesWarningCode				: WORD ; 						(* (NA) Internal Akuo Warning Code       	*)
	MesEventCode				: WORD ; 						(* (NA) Internal Akuo Event Code         	*)
	 
	MesCP_Read					: BOOL := TRUE; 						(* (NA) Permanent conditions for read		*)          

	MesCP_Write					: BOOL; 						(* (NA) Permanent conditions for read		*)    
                             						
END_STRUCT
END_TYPE

// ---- 01_Equipement_Library/Datalogger/Datalogger_IOWIT.TcDUT
TYPE Datalogger_IOWIT :		// Data from WIT in PTR
STRUCT
	

	MesData						: Datalogger ; 
		            			
	Transfo						: Transfo_MV ; 
	                			
	WS							: WS_PTR ; 
	                			
	MainMVCB					: MainMVCB_Sch ; 
	CB_INV						: ARRAY[1..CstNbInv_PTR_G] OF  TOR ; 
	CB_Transfo					: TOR ; 
	                				
	FSS							: FSS ; 
	DS							: TOR ; 
	MS	 						: TOR ; 





	MesInvReturnContact1 		: BOOL;		(* Inverter return contact 1 *)
	MesInvReturnContact2 		: BOOL;		(*  Inverter return contact 2 *)
	MesTransfoLocalTemp			: REAL;		(* (°C) Transformer room temperature *)
	

	MesAlarmCode				: WORD ; 	(* Internal Akuo Alarm Code *)
	MesWarningCode				: WORD ; 	(* Internal Akuo Warning Code *)
	MesEventCode				: WORD ; 	(* Internal Akuo Event Code *)
END_STRUCT
END_TYPE

// ---- 01_Equipement_Library/Datalogger/Datalogger_SchSkid.TcDUT
TYPE Datalogger_SchSkid :
STRUCT

	MesData							: Datalogger ; 							(* MesData *)
                        			                			
	MesComutLocal					: BOOL; 								(* FALSE := Local, TRUE := Remote (DI_204) *)
	MesState_MVCB					: BOOL; 								(* True := Fermé, False := Ouvert (DI_205) *)
	MesWatchdog_ProtectRelayVIP		: BOOL; 								(* WatchDog of VIP410 (DI_201)			   *)
	MesFault_ProtectRelayVIP		: BOOL; 								(* TRUE:= Fault, False:= OK, Déclenchement du défaut VIP (DI_206) *)
	                        			
	MesToggleRead					: BOOL; 								(* Cal State com of FB IO *)
	MesToggleWrite					: BOOL;;  								(* Cal State com of FB IO *)
	 
	DS_Synthesis					: TOR_Standard ; 								(* Synthesis of door sensors True = a door is opened (DI_209) 			 *)
	CB_INV							: ARRAY[1..CstNbInv_PTR_G] OF  TOR_Standard ; 	(* TRUE := CB opened, False : CB closed, INV 1 (DI_202) / INV 2 (DI_203) *)
	Transfo_Synthesis				: Transfo_MV; 							(* Transfo *)
	 	 						
END_STRUCT
END_TYPE

// ---- 01_Equipement_Library/Datalogger/Datalogger_Secu.TcDUT
TYPE Datalogger_Secu :
STRUCT
	
	MesData					: Datalogger ; 

	MesAlarm_Intrusion		: BOOL ;  (* Intrusion alarm *) 
	MesState_Siren1			: BOOL ; (* anti-intrusion siren is on *) 	                                                   			                                               
	MesState_Siren2			: BOOL ; (* anti-intrusion siren is on *) 	

	
END_STRUCT
END_TYPE

// ---- 01_Equipement_Library/Datalogger/Datalogger_SENECA.TcDUT
TYPE Datalogger_SENECA :
STRUCT
	
	MesData			: Datalogger ; 			  (* (NA) MesData *)
                        			                			                            	
	MesWindSp		: REAL ;				  (* (km/h) Wind speed of the weather station on SPP zone	 		*)
	MesWindDir		: REAL ;  				  (* (deg) Wind direction of the weather station on SPP zone	    *)
	 	 						
END_STRUCT
END_TYPE

// ---- 01_Equipement_Library/Fan/Fan_Standard.TcDUT
TYPE Fan_Standard :
STRUCT
	MesData : Fan;	(* (NA) Object fan	*)		
END_STRUCT
END_TYPE

// ---- 01_Equipement_Library/GRID/GRID.TcDUT
///////////
// Structure For DEIECommand. Main Operating Data to be saved (ex: OPC)  
//////////
TYPE GRID :
STRUCT
	// TC
	OUT_CmdAutCpl			 	: BOOL ;			(* (NA) Autorisation couplage (pulse)*)
	OUT_CmdDisconnect		 	: BOOL ;			(* (NA) Disconnect command (pulse)*)
	OUT_CmdEmergencyDisconnect	: BOOL ;			(* (NA) Emergency disconnect command (pulse)*)	
	OUT_SetptP 				 	: REAL ;			(* (kW) P Setpoint from EDF*)
	OUT_SetptQ 				 	: REAL ;			(* (kVar) Q Setpoint from EDF*)
	OUT_MesPPUnavailable		: BOOL ;			(* (NA) TS centrale indisponible*)
	OUT_MesPPConnected			: BOOL ; 			(* (NA)Centrale couplée(1)/Centrale Découplée(0)*)	
	
	// State 	
	MesAlarmCode				: WORD ; 			(* (NA) Internal Akuo Alarm Code*)
	MesWarningCode 			 	: WORD ; 			(* (NA) Internal Akuo Warning Code*)
	MesEventCode			 	: WORD ;			(* (NA) Internal Akuo Warning Code*)
	MesEventCode2				: WORD ; 			(* (NA) EventCode 2*)

	MesAlarmCom				 	: BOOL ;			(* (NA) Communication alarm *)
	MesCP_Read				 	: BOOL := TRUE; 	(* (NA) Cal : Read function enable*)
	
END_STRUCT
END_TYPE

// ---- 01_Equipement_Library/GRID/GRID_MADI.TcDUT
///////////
// Structure For DEIECommand. Main Operating Data to be saved (ex: OPC)  
//////////
TYPE GRID_MADI :
STRUCT
	// TC
	MesData					: GRID ;(* Object *)
	
END_STRUCT
END_TYPE

// ---- 01_Equipement_Library/GRID/GRID_Enedis.TcDUT
///////////
// Structure For DEIECommand. Main Operating Data to be saved (ex: OPC).
//////////
TYPE GRID_Enedis :
STRUCT
	
	MesData								: GRID ; 		(* GRID MesData *)
                                       	
	OUT_CmdPReg                         : BOOL ;     	(* (NA) Passage à P0 reçu DI*)
	OUT_CmdQReg	                   	    : BOOL ;     	(* (NA) Passage à Q0 reçu DI*)

	OUT_Rse								: BOOL; 		(* (NA) Protection en Rse(1) / Protection Hors RSE (O) *)
	OUT_TA								: BOOL; 		(* (NA) Telecaction en service (1) / Teleaction Hors service (0)*)
	
	MesEcart_HeureGrid					: DINT; 		(* (s) seconds of difference between EDF and SCADA times*)	
	
END_STRUCT
END_TYPE

// ---- 01_Equipement_Library/GRID/GRID_PLAN.TcDUT
///////////
// Structure For DEIECommand. Main Operating Data to be saved ( ex: OPC ) .  
//////////
TYPE GRID_PLAN :
STRUCT
	
	MesData			: GRID ; 

	//INPUT
                                       	
	OUT_CmdPReg                        	: BOOL ;     	(* Passage à P0 reçu DI*)
	OUT_CmdQReg	                    	: BOOL ;     	(* Passage à Q0 reçu DI*)

	OUT_Rse								: BOOL; (*Protection en Rse(1) / Protection Hors RSE (O) *)
	OUT_TA								: BOOL; (*Telecaction en service (1) / Teleaction Hors service (0)*)
          
	OUT_SetptU					: REAL ; (* (V) Voltage Setpoint from Grid*)
    OUT_SetptCosPhi          : REAL ;       (* (kW) Cosphi Setpoint from Grid*)           	                                                       
	//State                                             	                                                       

	
END_STRUCT
END_TYPE

// ---- 01_Equipement_Library/GRID/IEC104_PLAN.TcDUT
///////////
// Structure For DEIECommand. Main Operating Data to be saved ( ex: OPC ) .  
//////////
TYPE IEC104_PLAN :
STRUCT





	(* Double points *)
	(* 	Bit 0..1 = MesStartOn,
		Bit 2..3 = MesComTest_ON, 
		Bit 4..5 = MesCentraleCpl, 
		Bit 6..7 = MesCentrale_Ind*)
	OUT_MesLocal						: BOOL;
	OUT_MesDouble			AT%MB13		: BYTE;
	OUT_MesPosCB_SubMV					: BOOL; (*100*)
	OUT_MesPosSec_SubMV					: BOOL; (*101*)
	OUT_MesPosEarth_SubMV				: BOOL; (*102*)
	OUT_CmdPvF_On						: BOOL; (*103*)
	
	OUT_MesDouble2			AT%MB14		: BYTE; (**)
	OUT_CmdP							: UINT; (*105 - 0 : programado, 1: programado + regulacion primera*)
	OUT_CmdQ_On							: BOOL; (*107*)
	OUT_MesPosInter_33kV				: BOOL; (*106 - IT-PRC5020*)
	
	OUT_MesDouble3			AT%MB15		: BYTE; (**)
	OUT_MesPosSecLinea_33kV				: BOOL; (*108 - IT-PRC5021*)
	OUT_MesPosSec_33kV					: BOOL; (*109 - SC-PRC5025*)
	OUT_MesPosEarth_33kV				: BOOL; (*110 - SC-PRC5021*)
	OUT_MesPosInter_110kV				: BOOL; (*111 - IT-PRC7020*)	
                                                  
	OUT_MesDouble4			AT%MB16		: BYTE;
	OUT_MesPosSecLinea_110kV			: BOOL; (*112 - IT-PRC7027*)
 	
	
	
	(* Measured values, short floating point values *)
	OUT_MesP_33kV		 	AT%MB22		: REAL; (*IOA 1000*)
	OUT_MesQ_33kV			AT%MB26		: REAL; (*IOA 1001*)
	OUT_MesU12_33kV			AT%MB30		: REAL; (*IOA 1002*)
	OUT_MesI2_33kV 			AT%MB34		: REAL; (*IOA 1003*)
	OUT_MesP_110kV		 	AT%MB38		: REAL; (*IOA 1004*)
	OUT_MesQ_110kV			AT%MB42		: REAL; (*IOA 1005*)
	OUT_MesU12_110kV		AT%MB46		: REAL; (*IOA 1006*)
	OUT_MesI2_110kV 		AT%MB50		: REAL; (*IOA 1007*)
	OUT_SetptU				AT%MB54		: REAL; (*IOA 1008*)
	OUT_SetptPF				AT%MB58		: REAL; (*IOA 1009*)
	OUT_SetptQ				AT%MB62		: REAL; (*IOA 1010*)
	OUT_MesAvailability		AT%MB66		: REAL; (*IOA 1011*)
	OUT_MesPMax				AT%MB70		: REAL; (*IOA 1012*)
	OUT_MesGTI				AT%MB74		: REAL; (*IOA 1013*)
	OUT_MesTempPan			AT%MB82		: REAL; (*IOA 1014*)
	OUT_MesGHI				AT%MB86		: REAL; (*IOA 1015*)
	OUT_MesTempAmb			AT%MB90		: REAL; (*IOA 1016*)
	OUT_MesP_33kV_1			AT%MB94		: REAL; (*IOA 1017*)
	OUT_MesQ_33kV_1			AT%MB98		: REAL; (*IOA 1018*)
	OUT_MesU_33kV_1			AT%MB102	: REAL; (*IOA 1019*)
	OUT_MesI_33kV_1			AT%MB106	: REAL; (*IOA 1020*)
	OUT_MesTapPos			AT%MB110	: REAL; (*IOA 1021*)
	OUT_CmdQ				AT%MB114	: REAL; (*IOA 104 - 0 : desactivado, 1: QvU, 2: QvPF, 3: Q*)
	                                                     

	//TVC
	IN_SetptP1 				AT%MB150 	: REAL ;	(*IOA  CONSIGNE P*)
	IN_SetptU 				AT%MB154 	: REAL ;	(*IOA 1 CONSIGNE P*)
	IN_SetptPF 				AT%MB158 	: REAL ;	(*IOA 2 CONSIGNE P*)
	IN_SetptQ 				AT%MB162 	: REAL ;	(*IOA 3 CONSIGNE P*)
	IN_CmdQ 				AT%MB166 	: REAL ;	(*IOA 4 CONSIGNE P*)

	
END_STRUCT
END_TYPE

// ---- 01_Equipement_Library/GRID/IEC104_MADI.TcDUT
///////////
// Structure For DEIECommand. Main Operating Data to be saved ( ex: OPC ) .  
//////////
TYPE IEC104_MADI :
STRUCT

	(* Memory offset 0..99 unused *)
	(* Single points *)// MAx 8 bit per register . 0..7
	OUT_MesLocal			AT%MX10.0 	: BOOL;			(* IOA 12 BAT.LOCAL*)
	OUT_MesModeManuel_on	AT%MX10.1 	: BOOL; 		(* IOA 13 MANUAL*)
	OUT_MesModeAuto_on		AT%MX10.2 	: BOOL; 		(* IOA 14 AUTO*)
	OUT_MesCharging			AT%MX10.3 	: BOOL;			(* IOA 15 CHARGE.BAT*)
	OUT_MesDischarging		AT%MX10.4 	: BOOL;			(* IOA 16 DESCHARGE.BAT*)
	OUT_MesEs				AT%MX10.5 	: BOOL; 		(* IOA 20 ARRET.URGENCE*)
	OUT_MesToS				AT%MX10.6 	: BOOL; 		(* IOA 21 PRESENCE*)
	OUT_MesIncident			AT%MX10.7 	: BOOL;			(* IOA 19 INCIDENT*)
	OUT_MesFaultTeleMes		AT%MX11.0 	: BOOL;			(* IOA 37 DEFAUT CARTE TM*)
	OUT_MesFaultTeleCmd		AT%MX11.1 	: BOOL;			(* IOA 38 DEF FUNC TC*)
	OUT_MesFaultTeleSgnl	AT%MX11.2 	: BOOL;			(* IOA 39 DEF FONC TS*)
	OUT_MesIECServerFault	AT%MX11.3 	: BOOL;			(* IOA 41 DEF LIAISON 104*)
	
	(* Double points *)
	(* 	Bit 0..1 = MesStartOn,
		Bit 2..3 = MesComTest_ON, 
		Bit 4..5 = MesCentraleCpl, 
		Bit 6..7 = MesCentrale_Ind*)
	OUT_MesDouble			AT%MB12		: BYTE;
	MesDJOpen							: BOOL; 		(* IOA 51 DJ OPEN*)
	MesSoutirage_on						: BOOL;			(* IOA 43 ARRET.BAT*)
	MesComTest_on						: BOOL; 		(* IOA 44 TC.SOUTIRAGE *)
	MesCentrale_Cpl						: BOOL;			(* IOA 17 COUPL*)
	MesCentrale_indispo					: BOOL;			(* IOA 22 DISPO*)
	
	(* Measured values, short floating point values *)
	OUT_MesEconnected 		AT%MB42		: REAL;			(*IOA 5 NIVEAU BAT*)
	OUT_MesEmaxconnected 	AT%MB14		: REAL; 		(*IOA 6 STOCK MAX*)
	OUT_MesP 				AT%MB18		: REAL; 		(*IOA 1 P.ACTIVE*)
	OUT_MesQ 				AT%MB22		: REAL; 		(*IOA 2 P.REACTIVE*)
	OUT_MesU_HTA 			AT%MB26		: REAL; 		(*IOA 3 U.HTA*)
	OUT_MesFreq 			AT%MB30		: REAL; 		(*IOA 4 FREQUENCE*)
	OUT_MesPdispo_inj 		AT%MB34		: REAL; 		(*IOA 7 P.INJ MAX*)
	OUT_MesPdispo_abs 		AT%MB38		: REAL; 		(*IOA 8 P.SOUT MAX*)

	(*#################################################################*)
	(* TC *)
	IN_CmdModeManuel		AT%MX60.0 	: BOOL;			(* IOA 30 TC.MANUEL*)
	IN_CmdModeManuelOff		AT%MX60.1 	: BOOL;			(* Not implemented yet*)
	IN_CmdAut_Cpl			AT%MX60.2 	: BOOL; 		(* IOA 32 TC.COUPLAGE*)
	IN_CmdDisconnect		AT%MX60.3 	: BOOL;			(* IOA 33 TC.DECOUPLAGE*)
	IN_CmdConnect			AT%MX60.4 	: BOOL;			(* Not implemented*)
	
	(* TCD *)
	(* 	Bit 0..1 = command disconnecr,
		Bit 2..3 = command start, 
		Bit 4..5 =  command test, 
		Bit 6..7 = fourth double command *)
	IN_Cmddouble			AT%MB61		: BYTE;			(**)
	CmdSoutirage						: BOOL;			(* IOA 26 soutirage*)
	CmdTest								: BOOL;			(* IOA 27 TC.FICTIVE*)

	//TVC
	IN_SetptP 				AT%MB72 	: REAL ;		(*IOA 36 CONSIGNE P*)
	IN_ParamPmax 			AT%MB64 	: REAL ;    	(*IOA 34 CONSIGNE P+MAX *)
	IN_ParamPmin 			AT%MB68 	: REAL ;		(*IOA 35 CONSIGNE P-MAX *)

	
END_STRUCT
END_TYPE

// ---- 01_Equipement_Library/Fan/Fan.TcDUT
TYPE Fan :
STRUCT
		MesModeRun			: BOOL ;	(* (NA) Fan is running. 1 = running, 0 = not running (alarm) *)
		MesModeAuto			: BOOL ;	(* (NA) 1 = fan in in auto mode, 0 = fan is in manual mode 	 *)
		MesTemp				: REAL ; 	(* (C) Temperature // fTmp_Max	  							 *)
        MesStartTime 		: WORD ;	(* (Time) Cal: starting Time	  							 *)
        MesStopTime 		: WORD ;	(* (Time) Cal: stopping Time	  							 *)
		                                                                  							
		MesAlarmCode		: WORD ;    (* (NA) Internal Akuo AlarmCode   							 *)
		MesWarningCode		: WORD ;    (* (NA) Internal Akuo WarningCode 							 *)
		MesEventCode		: WORD ;    (* (NA) Internal Akuo EventCode   	 						 *)		
		
END_STRUCT
END_TYPE

// ---- 01_Equipement_Library/HVAC/HVAC.TcDUT
TYPE HVAC :
STRUCT

	MesSetptTemp		: REAL ;    	 (*(°C)  Temperature setpoint*)

	MesSetptHygro		: REAL ;    	 (*(%)   Hygrometry setpoint      *)

	MesOn				: BOOL ;    	 (*      HVAC is on *)

	MesAlarmCom			: BOOL ;    	 (*      Communication alarm *)

	MesWorkingHr 			: REAL ; 		 (* (s)	 Time AC has been on*)
	MesCP_Read			: BOOL := TRUE; (* 	 Read function enable*)
	MesCP_Write			: BOOL := FALSE; (* 	 Write function enable*)
	
	MesAlarmCode		: WORD ;		 (* 	 AlarmCode for the TGBT*)
	MesWarningCode		: WORD ;		 (* 	 WarningCode for the TGBT*)
	                                     

	
END_STRUCT
END_TYPE

// ---- 01_Equipement_Library/HVAC/HVAC_MADI.TcDUT
TYPE HVAC_MADI :
STRUCT
	MesData				: HVAC ;	

	MesHygro_Amb		: REAL ; 		 (*(%)	 Hygro value*)
	MesPressure1		: REAL ; 		 (*(bar) Pressure of the evaporatr 1 (bar )*)
	MesTemp_Room		: REAL ; 		 (*(°C)	 Temperature value .*)
	MesTemp_Outlet		: REAL ; 		 (*(°C)  Temperature at the HVAC output*)
	MesTemp_Outside		: REAL ; 		 (*(°C)  Outside air temperature*)
	
	MesSetptTempmin		: REAL ;    	 (*(°C)  Min Temperature setpoint *)
	MesSetptTempmax		: REAL ;    	 (*(°C)	 Max Temperature setpoint *)
	
	MesSetptHygromin	: REAL ;    	 (*(%)	 Min Hygrometry setpoint  *)
	MesSetptHygromax	: REAL ;    	 (*(%)	 Max Hygrometry setpoint  *)
	
	MesAlarmsSynthesis	: BOOL ;         (*      Alamrs synthesis *)
	
	MesCooling			: BOOL ;   		 (*()	 The HVAC is cooling the air*)
	MesHeating			: BOOL ; 		 (*()	 The HVAC is heating the air*)
	                                     
	MesAlarm1			: WORD ; 		 (* 	 HVAC Alarm word 1*)
	MesAlarm2			: WORD ; 		 (* 	 HVAC Alarm word 2*)
	MesAlarm3			: WORD ; 		 (* 	 HVAC Alarm word 3*)
	
END_STRUCT
END_TYPE

// ---- 01_Equipement_Library/HVAC/HVAC_MeAcMbs1.TcDUT
TYPE HVAC_MeAcMbs1 :
STRUCT
	MesData : HVAC;						(* (NA) Main Structure*)
	
	IN_SetptTemp		: REAL ;		(* (°C) Temperature setpoint input *)
	IN_CmdStatus		: BOOL ;		(* (NA) Status order: 1= On, 0= Off*)
	
	MesMode				: INT  ;		(* (NA) AC Unit Mode : 0:Auto, 1: Heat, 2: Dry, 3: Fan, 4: Cool*)
	MesFanMode			: WORD ;		(* (NA) Fan Speed (0:Auto, 1:Low, 2:Mid1, 3:Mid2, 4:High) *)
	MesTempRef			: REAL ;		(* (°C) Temperature reference: Used to update the measured temp for PID of the HVAC*)
	MesbAlarm			: BOOL ;		(* (NA) Alarm condition*)
	MesErrorCode		: WORD ; 		(* (NA) Error Code*)
	MesTempRoom			: REAL ; 		(* (°C)	Temperature value *)
 	MesTempRealSetpt	: REAL ;		(* (°C) Real temperature setpoint if a temp ref is entered *)
	
	MesAlarm1 			: WORD;			(* (NA) Alarm *)
	MesAlarm2 			: WORD;         (* (NA) Alarm *)
	MesAlarm3 			: WORD;         (* (NA) Alarm *)
	MesAlarm4 			: WORD;         (* (NA) Alarm *)
	
END_STRUCT
END_TYPE

// ---- 01_Equipement_Library/HVAC/HVAC_NARADA.TcDUT
TYPE HVAC_NARADA :
STRUCT
	
	MesData				: HVAC ;	

	MesCoolTemp			: REAL	;		(*(°C)	Cooling Temperature value .*)
	MesCoolSens			: REAL	;		(*(°C)	Cooling Sensitivity value .*)
	MesHeatingTemp		: REAL	;		(*(°C)	Cooling Temperature value .*)
	MesHeatingSens		: REAL	;		(*(°C)	Cooling Sensitivity value .*)
	MesSetptHygro		: REAL ;		(*(%)	 Hygrometry setpoint  *)
	MesSensHygro		: REAL ;		(*(%)	 Hygrometry sensitivity  *)
	MesTempmin			: REAL ;		(*(°C)  Min Temperature *)
	MesTempmax			: REAL ;		(*(°C)	 Max Temperature *)
	MesHygromax			: REAL ;		(*(%)	 Maximum humidity*)
	MesState			: REAL ;		(* status of HVAC*)
	MesStateFanInternal	: BOOL ;		(* Status of fan internal*)
	MesStateFanExternal	: BOOL ;		(*Status of fan external*)
	MesCompressorStatus : BOOL ;		(* State of compressor*)
	MesHeating			: REAL ;		(*()	 The HVAC is heating the air*)
	MesFrostTemp		: BOOL ;		(* (°C)frosting temperature *)
	MesCondTemp			: BOOL ;		(* (°C Condescending temperature *)	
	MesPressure1		: REAL ; 		 (*(bar) Pressure of the evaporatr 1 (bar )*)
	MesTemp_Room		: REAL ; 		 (*(°C)	 Temperature value .*)
	MesHygro			: REAL ; 		 (*(%) Humidity of the hvac *)
	MesTemp_Outside		: REAL ; 		 (*(°C)  Outside air temperature*)
	                                     
	MesAlarmLow			: WORD ; 		 (* 	 HVAC Alarm word 1*)
	MesAlarmHigh		: WORD ; 		 (* 	 HVAC Alarm word 2*)
	
END_STRUCT
END_TYPE

// ---- 01_Equipement_Library/HVAC/HVAC_Standard.TcDUT
TYPE HVAC_Standard :
STRUCT
	MesData				: HVAC ;	

	MesHygro_Amb		: REAL ; 		 (*(%)	 Hygro value*)
	MesPressure1		: REAL ; 		 (*(bar) Pressure of the evaporatr 1 (bar )*)
	MesTemp_Room		: REAL ; 		 (*(°C)	 Temperature value .*)
	MesTemp_Outlet		: REAL ; 		 (*(°C)  Temperature at the HVAC output*)
	MesTemp_Outside		: REAL ; 		 (*(°C)  Outside air temperature*)
	
	MesSetptTempmin		: REAL ;    	 (*(°C)  Min Temperature setpoint *)
	MesSetptTempmax		: REAL ;    	 (*(°C)	 Max Temperature setpoint *)
	
	MesSetptHygromin	: REAL ;    	 (*(%)	 Min Hygrometry setpoint  *)
	MesSetptHygromax	: REAL ;    	 (*(%)	 Max Hygrometry setpoint  *)
	
	MesAlarmsSynthesis	: BOOL ;         (*      Alamrs synthesis *)
	
	MesCooling			: BOOL ;   		 (*()	 The HVAC is cooling the air*)
	MesHeating			: BOOL ; 		 (*()	 The HVAC is heating the air*)
	                                     
	MesAlarm1			: WORD ; 		 (* 	 HVAC Alarm word 1*)
	MesAlarm2			: WORD ; 		 (* 	 HVAC Alarm word 2*)
	MesAlarm3			: WORD ; 		 (* 	 HVAC Alarm word 3*)
	
END_STRUCT
END_TYPE

// ---- 01_Equipement_Library/HVAC/HVAC_SAFT.TcDUT
TYPE HVAC_SAFT :
STRUCT
	MesData				: HVAC ;	

	MesHygro_Amb		: REAL ; 		 (*(%)	 Hygro value*)
	MesTemp_Room		: REAL ; 		 (*(°C)	 Temperature value .*)
	MesTemp_Outside		: REAL ; 		 (*(°C)  Outside air temperature*)
	
	MesIDState			: WORD ; (* (NA) SubBankHVAC_St [SubBankHVAC_St] *) 

	
END_STRUCT
END_TYPE

// ---- 01_Equipement_Library/Inverter/INV.TcDUT
///////////
// Structure For Inverter. Main Operating Data to be saved (ex: OPC).  
//////////
TYPE INV :
STRUCT
	
